LIN {X 0,Y 250.024,Z 759.381,A -85,B 0,C 180,E1 17271.33,E2 17271.33} C_VEL
LIN {X 0,Y 248.705,Z 752.621,A -85,B 0,C 180,E1 17277.4,E2 17277.4} C_VEL
LIN {X 0,Y 248.828,Z 740.046,A -85,B 0,C 180,E1 17283.485,E2 17283.485} C_VEL
LIN {X 0,Y 250.046,Z 721.857,A -85,B 0,C 180,E1 17289.123,E2 17289.123} C_VEL
LIN {X 0,Y 252.287,Z 698.147,A -85,B 0,C 180,E1 17294.071,E2 17294.071} C_VEL
LIN {X 0,Y 254.747,Z 670.659,A -85,B 0,C 180,E1 17297.96,E2 17297.96} C_VEL
LIN {X 0,Y 256.815,Z 639.717,A -85,B 0,C 180,E1 17300.765,E2 17300.765} C_VEL
LIN {X 0,Y 257.718,Z 620.09,A -85,B 0,C 180,E1 17301.928,E2 17301.928} C_VEL
LIN {X 0,Y 260.308,Z 616.482,A -85,B 0,C 180,E1 17302.928,E2 17302.928} C_VEL
LIN {X 0,Y 264.834,Z 607.073,A -85,B 0,C 180,E1 17303.896,E2 17303.896} C_VEL
LIN {X 0,Y 272.961,Z 594.621,A -85,B 0,C 180,E1 17306.378,E2 17306.378} C_VEL
LIN {X 0,Y 281.526,Z 610.071,A -85,B 0,C 180,E1 17312.421,E2 17312.421} C_VEL
LIN {X 0,Y 291.528,Z 631.973,A -85,B 0,C 180,E1 17318.409,E2 17318.409} C_VEL
LIN {X 0,Y 298.079,Z 654.366,A -85,B 0,C 180,E1 17323.266,E2 17323.266} C_VEL
LIN {X 0,Y 299.11,Z 663.186,A -85,B 0,C 180,E1 17324.88,E2 17324.88} C_VEL
LIN {X 0,Y 288.395,Z 696.037,A -85,B 0,C 180,E1 17328.65,E2 17328.65} C_VEL
LIN {X 0,Y 277.431,Z 723.704,A -85,B 0,C 180,E1 17333.247,E2 17333.247} C_VEL
LIN {X 0,Y 266.011,Z 748.871,A -85,B 0,C 180,E1 17339.297,E2 17339.297} C_VEL
LIN {X 0,Y 256.342,Z 769.366,A -85,B 0,C 180,E1 17346.585,E2 17346.585} C_VEL
LIN {X 0,Y 249.921,Z 783.871,A -85,B 0,C 180,E1 17354.413,E2 17354.413} C_VEL
LIN {X 0,Y 246.587,Z 793.255,A -85,B 0,C 180,E1 17362.97,E2 17362.97} C_VEL
LIN {X 0,Y 245.826,Z 796.854,A -85,B 0,C 180,E1 17370.001,E2 17370.001} C_VEL
LIN {X 0,Y 245.618,Z 797.004,A -85,B 0,C 180,E1 17377.059,E2 17377.059} C_VEL
LIN {X 0,Y 246.956,Z 793.586,A -85,B 0,C 180,E1 17384.15,E2 17384.15} C_VEL
LIN {X 0,Y 251.318,Z 784.05,A -85,B 0,C 180,E1 17392.976,E2 17392.976} C_VEL
LIN {X 0,Y 258.612,Z 769.768,A -85,B 0,C 180,E1 17400.706,E2 17400.706} C_VEL
LIN {X 0,Y 269.525,Z 749.005,A -85,B 0,C 180,E1 17408.021,E2 17408.021} C_VEL
LIN {X 0,Y 282.105,Z 723.317,A -85,B 0,C 180,E1 17414.065,E2 17414.065} C_VEL
LIN {X 0,Y 294.764,Z 693.635,A -85,B 0,C 180,E1 17418.777,E2 17418.777} C_VEL
LIN {X 0,Y 304.453,Z 665.385,A -85,B 0,C 180,E1 17421.913,E2 17421.913} C_VEL
LIN {X 0,Y 299.008,Z 642.776,A -85,B 0,C 180,E1 17427.136,E2 17427.136} C_VEL
LIN {X 0,Y 298.518,Z 641.319,A -85,B 0,C 180,E1 17427.506,E2 17427.506} C_VEL
LIN {X 0,Y 282.147,Z 661.718,A -85,B 0,C 180,E1 17429.533,E2 17429.533} C_VEL
LIN {X 0,Y 270.306,Z 673.201,A -85,B 0,C 180,E1 17431.601,E2 17431.601} C_VEL
LIN {X 0,Y 261.762,Z 680.494,A -85,B 0,C 180,E1 17433.454,E2 17433.454} C_VEL
LIN {X 0,Y 258.089,Z 683.189,A -85,B 0,C 180,E1 17434.447,E2 17434.447} C_VEL
LIN {X 0,Y 253.572,Z 685.97,A -85,B 0,C 180,E1 17435.932,E2 17435.932} C_VEL
LIN {X 0,Y 252.951,Z 690.362,A -85,B 0,C 180,E1 17436.705,E2 17436.705} C_VEL
LIN {X 0,Y 250.934,Z 714.808,A -85,B 0,C 180,E1 17440.677,E2 17440.677} C_VEL
LIN {X 0,Y 249.341,Z 734.383,A -85,B 0,C 180,E1 17445.567,E2 17445.567} C_VEL
LIN {X 0,Y 248.688,Z 747.033,A -85,B 0,C 180,E1 17450.386,E2 17450.386} C_VEL
LIN {X 0,Y 248.844,Z 754.316,A -85,B 0,C 180,E1 17454.773,E2 17454.773} C_VEL
LIN {X 0,Y 250.011,Z 758.572,A -85,B 0,C 180,E1 17459.992,E2 17459.992} C_VEL
LIN {X 0,Y 251.473,Z 758.815,A -85,B 0,C 180,E1 17463.432,E2 17463.432} C_VEL
LIN {X 0,Y 255.403,Z 754.257,A -85,B 0,C 180,E1 17469.343,E2 17469.343} C_VEL
LIN {X 0,Y 260.605,Z 743.743,A -85,B 0,C 180,E1 17474.667,E2 17474.667} C_VEL
LIN {X 0,Y 266.042,Z 728.772,A -85,B 0,C 180,E1 17479.027,E2 17479.027} C_VEL
LIN {X 0,Y 271.609,Z 707.895,A -85,B 0,C 180,E1 17482.879,E2 17482.879} C_VEL
LIN {X 0,Y 276.132,Z 682.599,A -85,B 0,C 180,E1 17485.787,E2 17485.787} C_VEL
LIN {X 0,Y 276.83,Z 677.028,A -85,B 0,C 180,E1 17486.267,E2 17486.267} C_VEL
LIN {X 0,Y 282.767,Z 670.413,A -85,B 0,C 180,E1 17487.132,E2 17487.132} C_VEL
LIN {X 0,Y 299.288,Z 647.276,A -85,B 0,C 180,E1 17488.81,E2 17488.81} C_VEL
LIN {X 0,Y 301.073,Z 645.58,A -85,B 0,C 180,E1 17489.104,E2 17489.104} C_VEL
LIN {X 0,Y 309.235,Z 670.823,A -85,B 0,C 180,E1 17494.629,E2 17494.629} C_VEL
LIN {X 0,Y 308.878,Z 675.554,A -85,B 0,C 180,E1 17495.18,E2 17495.18} C_VEL
LIN {X 0,Y 296.991,Z 714.596,A -85,B 0,C 180,E1 17498.62,E2 17498.62} C_VEL
LIN {X 0,Y 284.585,Z 746.683,A -85,B 0,C 180,E1 17502.891,E2 17502.891} C_VEL
LIN {X 0,Y 272.037,Z 774.342,A -85,B 0,C 180,E1 17508.261,E2 17508.261} C_VEL
LIN {X 0,Y 260.443,Z 798.326,A -85,B 0,C 180,E1 17515.094,E2 17515.094} C_VEL
LIN {X 0,Y 251.52,Z 817.448,A -85,B 0,C 180,E1 17523.159,E2 17523.159} C_VEL
LIN {X 0,Y 246.513,Z 831.268,A -85,B 0,C 180,E1 17532.175,E2 17532.175} C_VEL
LIN {X 0,Y 245.059,Z 838.394,A -85,B 0,C 180,E1 17540.101,E2 17540.101} C_VEL
LIN {X 0,Y 244.928,Z 841.087,A -85,B 0,C 180,E1 17546.467,E2 17546.467} C_VEL
LIN {X 0,Y 245.399,Z 841.461,A -85,B 0,C 180,E1 17549.999,E2 17549.999} C_VEL
LIN {X 0,Y 244.964,Z 839.528,A -85,B 0,C 180,E1 17557.077,E2 17557.077} C_VEL
LIN {X 0,Y 246.082,Z 832.265,A -85,B 0,C 180,E1 17566.02,E2 17566.02} C_VEL
LIN {X 0,Y 250.068,Z 819.039,A -85,B 0,C 180,E1 17574.989,E2 17574.989} C_VEL
LIN {X 0,Y 258.016,Z 799.995,A -85,B 0,C 180,E1 17583.254,E2 17583.254} C_VEL
LIN {X 0,Y 268.824,Z 775.778,A -85,B 0,C 180,E1 17590.32,E2 17590.32} C_VEL
LIN {X 0,Y 280.754,Z 747.171,A -85,B 0,C 180,E1 17596.004,E2 17596.004} C_VEL
LIN {X 0,Y 292.476,Z 715.007,A -85,B 0,C 180,E1 17600.354,E2 17600.354} C_VEL
LIN {X 0,Y 297.708,Z 697.847,A -85,B 0,C 180,E1 17602.086,E2 17602.086} C_VEL
LIN {X 0,Y 281.447,Z 707.401,A -85,B 0,C 180,E1 17604.084,E2 17604.084} C_VEL
LIN {X 0,Y 276.293,Z 721.227,A -85,B 0,C 180,E1 17606.569,E2 17606.569} C_VEL
LIN {X 0,Y 268.734,Z 733.756,A -85,B 0,C 180,E1 17608.644,E2 17608.644} C_VEL
LIN {X 0,Y 261.291,Z 743.898,A -85,B 0,C 180,E1 17610.882,E2 17610.882} C_VEL
LIN {X 0,Y 260.962,Z 744.422,A -85,B 0,C 180,E1 17611.073,E2 17611.073} C_VEL
LIN {X 0,Y 253.58,Z 755.494,A -85,B 0,C 180,E1 17616.325,E2 17616.325} C_VEL
LIN {X 0,Y 247.612,Z 761.565,A -85,B 0,C 180,E1 17622.267,E2 17622.267} C_VEL
LIN {X 0,Y 245.037,Z 762.531,A -85,B 0,C 180,E1 17625.748,E2 17625.748} C_VEL
LIN {X 0,Y 242.317,Z 760.769,A -85,B 0,C 180,E1 17631.052,E2 17631.052} C_VEL
LIN {X 0,Y 240.885,Z 753.621,A -85,B 0,C 180,E1 17637.315,E2 17637.315} C_VEL
LIN {X 0,Y 240.963,Z 740.642,A -85,B 0,C 180,E1 17643.599,E2 17643.599} C_VEL
LIN {X 0,Y 242.241,Z 721.934,A -85,B 0,C 180,E1 17649.42,E2 17649.42} C_VEL
LIN {X 0,Y 244.575,Z 697.686,A -85,B 0,C 180,E1 17654.525,E2 17654.525} C_VEL
LIN {X 0,Y 247.222,Z 668.633,A -85,B 0,C 180,E1 17658.594,E2 17658.594} C_VEL
LIN {X 0,Y 249.103,Z 641.736,A -85,B 0,C 180,E1 17661.109,E2 17661.109} C_VEL
LIN {X 0,Y 251.183,Z 639.486,A -85,B 0,C 180,E1 17662.063,E2 17662.063} C_VEL
LIN {X 0,Y 256.836,Z 628.431,A -85,B 0,C 180,E1 17663.259,E2 17663.259} C_VEL
LIN {X 0,Y 258.62,Z 624.905,A -85,B 0,C 180,E1 17663.659,E2 17663.659} C_VEL
LIN {X 0,Y 264.07,Z 614.767,A -85,B 0,C 180,E1 17664.935,E2 17664.935} C_VEL
LIN {X 0,Y 271.122,Z 603.638,A -85,B 0,C 180,E1 17666.882,E2 17666.882} C_VEL
LIN {X 0,Y 279.782,Z 620.232,A -85,B 0,C 180,E1 17673.047,E2 17673.047} C_VEL
LIN {X 0,Y 288.455,Z 642.214,A -85,B 0,C 180,E1 17678.895,E2 17678.895} C_VEL
LIN {X 0,Y 293.409,Z 663.904,A -85,B 0,C 180,E1 17683.625,E2 17683.625} C_VEL
LIN {X 0,Y 283.073,Z 696.013,A -85,B 0,C 180,E1 17687.436,E2 17687.436} C_VEL
LIN {X 0,Y 271.188,Z 724.764,A -85,B 0,C 180,E1 17692.255,E2 17692.255} C_VEL
LIN {X 0,Y 259.284,Z 749.835,A -85,B 0,C 180,E1 17698.41,E2 17698.41} C_VEL
LIN {X 0,Y 249.135,Z 770.237,A -85,B 0,C 180,E1 17705.865,E2 17705.865} C_VEL
LIN {X 0,Y 242.475,Z 784.438,A -85,B 0,C 180,E1 17713.736,E2 17713.736} C_VEL
LIN {X 0,Y 238.773,Z 794.017,A -85,B 0,C 180,E1 17722.738,E2 17722.738} C_VEL
LIN {X 0,Y 237.977,Z 797.575,A -85,B 0,C 180,E1 17730.001,E2 17730.001} C_VEL
LIN {X 0,Y 237.764,Z 797.7,A -85,B 0,C 180,E1 17737.294,E2 17737.294} C_VEL
LIN {X 0,Y 239.24,Z 794.261,A -85,B 0,C 180,E1 17744.616,E2 17744.616} C_VEL
LIN {X 0,Y 243.928,Z 784.719,A -85,B 0,C 180,E1 17753.714,E2 17753.714} C_VEL
LIN {X 0,Y 251.718,Z 770.414,A -85,B 0,C 180,E1 17761.643,E2 17761.643} C_VEL
LIN {X 0,Y 263.246,Z 749.644,A -85,B 0,C 180,E1 17769.097,E2 17769.097} C_VEL
LIN {X 0,Y 276.418,Z 723.92,A -85,B 0,C 180,E1 17775.217,E2 17775.217} C_VEL
LIN {X 0,Y 289.272,Z 695.04,A -85,B 0,C 180,E1 17779.849,E2 17779.849} C_VEL
LIN {X 0,Y 298.783,Z 668.445,A -85,B 0,C 180,E1 17782.891,E2 17782.891} C_VEL
LIN {X 0,Y 295.453,Z 652.057,A -85,B 0,C 180,E1 17786.775,E2 17786.775} C_VEL
LIN {X 0,Y 280.732,Z 668.46,A -85,B 0,C 180,E1 17788.597,E2 17788.597} C_VEL
LIN {X 0,Y 268.852,Z 679.276,A -85,B 0,C 180,E1 17790.577,E2 17790.577} C_VEL
LIN {X 0,Y 260.135,Z 686.335,A -85,B 0,C 180,E1 17792.341,E2 17792.341} C_VEL
LIN {X 0,Y 247.479,Z 695.108,A -85,B 0,C 180,E1 17795.816,E2 17795.816} C_VEL
LIN {X 0,Y 244.805,Z 696.846,A -85,B 0,C 180,E1 17797.215,E2 17797.215} C_VEL
LIN {X 0,Y 242.653,Z 719.9,A -85,B 0,C 180,E1 17801.406,E2 17801.406} C_VEL
LIN {X 0,Y 241.28,Z 738.13,A -85,B 0,C 180,E1 17806.427,E2 17806.427} C_VEL
LIN {X 0,Y 240.793,Z 750.869,A -85,B 0,C 180,E1 17811.886,E2 17811.886} C_VEL
LIN {X 0,Y 241.623,Z 758.616,A -85,B 0,C 180,E1 17817.97,E2 17817.97} C_VEL
LIN {X 0,Y 243.765,Z 760.451,A -85,B 0,C 180,E1 17823.541,E2 17823.541} C_VEL
LIN {X 0,Y 247.928,Z 756.572,A -85,B 0,C 180,E1 17829.627,E2 17829.627} C_VEL
LIN {X 0,Y 253.445,Z 746.827,A -85,B 0,C 180,E1 17835.091,E2 17835.091} C_VEL
LIN {X 0,Y 259.82,Z 731.185,A -85,B 0,C 180,E1 17839.943,E2 17839.943} C_VEL
LIN {X 0,Y 265.992,Z 710.335,A -85,B 0,C 180,E1 17843.945,E2 17843.945} C_VEL
LIN {X 0,Y 270.352,Z 689.796,A -85,B 0,C 180,E1 17846.514,E2 17846.514} C_VEL
LIN {X 0,Y 276.719,Z 683.522,A -85,B 0,C 180,E1 17847.48,E2 17847.48} C_VEL
LIN {X 0,Y 292.53,Z 664.243,A -85,B 0,C 180,E1 17849.263,E2 17849.263} C_VEL
LIN {X 0,Y 297.533,Z 656.963,A -85,B 0,C 180,E1 17849.663,E2 17849.663} C_VEL
LIN {X 0,Y 300.096,Z 661.994,A -85,B 0,C 180,E1 17851.101,E2 17851.101} C_VEL
LIN {X 0,Y 303.842,Z 675.889,A -85,B 0,C 180,E1 17854.044,E2 17854.044} C_VEL
LIN {X 0,Y 291.982,Z 713.613,A -85,B 0,C 180,E1 17857.373,E2 17857.373} C_VEL
LIN {X 0,Y 279.227,Z 745.459,A -85,B 0,C 180,E1 17861.604,E2 17861.604} C_VEL
LIN {X 0,Y 265.928,Z 773.501,A -85,B 0,C 180,E1 17867.076,E2 17867.076} C_VEL
LIN {X 0,Y 253.719,Z 797.558,A -85,B 0,C 180,E1 17874.027,E2 17874.027} C_VEL
LIN {X 0,Y 244.173,Z 816.877,A -85,B 0,C 180,E1 17882.382,E2 17882.382} C_VEL
LIN {X 0,Y 238.791,Z 830.549,A -85,B 0,C 180,E1 17891.578,E2 17891.578} C_VEL
LIN {X 0,Y 237.146,Z 837.999,A -85,B 0,C 180,E1 17900.254,E2 17900.254} C_VEL
LIN {X 0,Y 237.044,Z 840.385,A -85,B 0,C 180,E1 17906.349,E2 17906.349} C_VEL
LIN {X 0,Y 237.516,Z 840.75,A -85,B 0,C 180,E1 17909.999,E2 17909.999} C_VEL
LIN {X 0,Y 237.073,Z 838.786,A -85,B 0,C 180,E1 17917.314,E2 17917.314} C_VEL
LIN {X 0,Y 237.855,Z 833.399,A -85,B 0,C 180,E1 17924.702,E2 17924.702} C_VEL
LIN {X 0,Y 241.457,Z 821.32,A -85,B 0,C 180,E1 17933.97,E2 17933.97} C_VEL
LIN {X 0,Y 248.933,Z 803.637,A -85,B 0,C 180,E1 17942.536,E2 17942.536} C_VEL
LIN {X 0,Y 259.384,Z 781.296,A -85,B 0,C 180,E1 17949.792,E2 17949.792} C_VEL
LIN {X 0,Y 271.8,Z 753.577,A -85,B 0,C 180,E1 17955.918,E2 17955.918} C_VEL
LIN {X 0,Y 284.241,Z 722.074,A -85,B 0,C 180,E1 17960.616,E2 17960.616} C_VEL
LIN {X 0,Y 287.935,Z 711.502,A -85,B 0,C 180,E1 17961.832,E2 17961.832} C_VEL
LIN {X 0,Y 287.56,Z 710.09,A -85,B 0,C 180,E1 17962.155,E2 17962.155} C_VEL
LIN {X 0,Y 274.608,Z 716.397,A -85,B 0,C 180,E1 17963.919,E2 17963.919} C_VEL
LIN {X 0,Y 264.992,Z 737.124,A -85,B 0,C 180,E1 17968.679,E2 17968.679} C_VEL
LIN {X 0,Y 260.962,Z 744.422,A -85,B 0,C 180,E1 17971.073,E2 17971.073} C_VEL
LIN {X 0,Y 252.831,Z 753.354,A -85,B 0,C 180,E1 17973.932,E2 17973.932} C_VEL
LIN {X 0,Y 245.199,Z 759.728,A -85,B 0,C 180,E1 17976.926,E2 17976.926} C_VEL
LIN {X 0,Y 244.902,Z 759.939,A -85,B 0,C 180,E1 17977.162,E2 17977.162} C_VEL
LIN {X 0,Y 240.338,Z 763.539,A -85,B 0,C 180,E1 17981.712,E2 17981.712} C_VEL
LIN {X 0,Y 237.568,Z 764.279,A -85,B 0,C 180,E1 17985.29,E2 17985.29} C_VEL
LIN {X 0,Y 234.625,Z 762.124,A -85,B 0,C 180,E1 17990.756,E2 17990.756} C_VEL
LIN {X 0,Y 233.035,Z 754.61,A -85,B 0,C 180,E1 17997.225,E2 17997.225} C_VEL
LIN {X 0,Y 233.093,Z 741.101,A -85,B 0,C 180,E1 18003.72,E2 18003.72} C_VEL
LIN {X 0,Y 234.445,Z 721.899,A -85,B 0,C 180,E1 18009.736,E2 18009.736} C_VEL
LIN {X 0,Y 236.758,Z 698.18,A -85,B 0,C 180,E1 18014.779,E2 18014.779} C_VEL
LIN {X 0,Y 239.462,Z 669.534,A -85,B 0,C 180,E1 18018.897,E2 18018.897} C_VEL
LIN {X 0,Y 240.33,Z 659.681,A -85,B 0,C 180,E1 18020.072,E2 18020.072} C_VEL
LIN {X 0,Y 243.745,Z 655.911,A -85,B 0,C 180,E1 18021.494,E2 18021.494} C_VEL
LIN {X 0,Y 248.777,Z 647.551,A -85,B 0,C 180,E1 18022.619,E2 18022.619} C_VEL
LIN {X 0,Y 254.503,Z 639.221,A -85,B 0,C 180,E1 18024.229,E2 18024.229} C_VEL
LIN {X 0,Y 260.251,Z 628.282,A -85,B 0,C 180,E1 18025.326,E2 18025.326} C_VEL
LIN {X 0,Y 267.14,Z 616.064,A -85,B 0,C 180,E1 18026.874,E2 18026.874} C_VEL
LIN {X 0,Y 269.344,Z 613.016,A -85,B 0,C 180,E1 18027.512,E2 18027.512} C_VEL
LIN {X 0,Y 277.59,Z 630.287,A -85,B 0,C 180,E1 18033.585,E2 18033.585} C_VEL
LIN {X 0,Y 284.434,Z 650.554,A -85,B 0,C 180,E1 18038.986,E2 18038.986} C_VEL
LIN {X 0,Y 287.585,Z 668.623,A -85,B 0,C 180,E1 18042.956,E2 18042.956} C_VEL
LIN {X 0,Y 275.911,Z 700.839,A -85,B 0,C 180,E1 18046.865,E2 18046.865} C_VEL
LIN {X 0,Y 263.358,Z 729.318,A -85,B 0,C 180,E1 18051.974,E2 18051.974} C_VEL
LIN {X 0,Y 251.216,Z 753.431,A -85,B 0,C 180,E1 18058.288,E2 18058.288} C_VEL
LIN {X 0,Y 240.94,Z 773.175,A -85,B 0,C 180,E1 18066.059,E2 18066.059} C_VEL
LIN {X 0,Y 233.81,Z 787.611,A -85,B 0,C 180,E1 18075.038,E2 18075.038} C_VEL
LIN {X 0,Y 230.969,Z 794.774,A -85,B 0,C 180,E1 18082.492,E2 18082.492} C_VEL
LIN {X 0,Y 230.122,Z 798.296,A -85,B 0,C 180,E1 18090.001,E2 18090.001} C_VEL
LIN {X 0,Y 229.925,Z 798.396,A -85,B 0,C 180,E1 18097.544,E2 18097.544} C_VEL
LIN {X 0,Y 231.529,Z 794.941,A -85,B 0,C 180,E1 18105.114,E2 18105.114} C_VEL
LIN {X 0,Y 236.582,Z 785.381,A -85,B 0,C 180,E1 18114.498,E2 18114.498} C_VEL
LIN {X 0,Y 244.907,Z 771.067,A -85,B 0,C 180,E1 18122.63,E2 18122.63} C_VEL
LIN {X 0,Y 257.095,Z 750.279,A -85,B 0,C 180,E1 18130.22,E2 18130.22} C_VEL
LIN {X 0,Y 270.864,Z 724.529,A -85,B 0,C 180,E1 18136.413,E2 18136.413} C_VEL
LIN {X 0,Y 284.529,Z 694.748,A -85,B 0,C 180,E1 18141.199,E2 18141.199} C_VEL
LIN {X 0,Y 293.095,Z 671.056,A -85,B 0,C 180,E1 18144.012,E2 18144.012} C_VEL
LIN {X 0,Y 291.882,Z 663.652,A -85,B 0,C 180,E1 18145.821,E2 18145.821} C_VEL
LIN {X 0,Y 290.566,Z 663.826,A -85,B 0,C 180,E1 18146.205,E2 18146.205} C_VEL
LIN {X 0,Y 273.557,Z 680.347,A -85,B 0,C 180,E1 18148.387,E2 18148.387} C_VEL
LIN {X 0,Y 258.118,Z 692.28,A -85,B 0,C 180,E1 18151.287,E2 18151.287} C_VEL
LIN {X 0,Y 244.499,Z 701.239,A -85,B 0,C 180,E1 18154.894,E2 18154.894} C_VEL
LIN {X 0,Y 236.5,Z 705.475,A -85,B 0,C 180,E1 18157.975,E2 18157.975} C_VEL
LIN {X 0,Y 233.928,Z 731.79,A -85,B 0,C 180,E1 18164.079,E2 18164.079} C_VEL
LIN {X 0,Y 233.019,Z 747.465,A -85,B 0,C 180,E1 18169.733,E2 18169.733} C_VEL
LIN {X 0,Y 233.262,Z 756.973,A -85,B 0,C 180,E1 18175.353,E2 18175.353} C_VEL
LIN {X 0,Y 234.413,Z 761.088,A -85,B 0,C 180,E1 18179.992,E2 18179.992} C_VEL
LIN {X 0,Y 236.034,Z 762.072,A -85,B 0,C 180,E1 18183.657,E2 18183.657} C_VEL
LIN {X 0,Y 239.713,Z 759.701,A -85,B 0,C 180,E1 18189.046,E2 18189.046} C_VEL
LIN {X 0,Y 244.85,Z 752.504,A -85,B 0,C 180,E1 18194.264,E2 18194.264} C_VEL
LIN {X 0,Y 251.283,Z 739.619,A -85,B 0,C 180,E1 18199.278,E2 18199.278} C_VEL
LIN {X 0,Y 258.195,Z 720.933,A -85,B 0,C 180,E1 18203.683,E2 18203.683} C_VEL
LIN {X 0,Y 264.036,Z 700.867,A -85,B 0,C 180,E1 18206.797,E2 18206.797} C_VEL
LIN {X 0,Y 278.176,Z 687.826,A -85,B 0,C 180,E1 18208.816,E2 18208.816} C_VEL
LIN {X 0,Y 295.409,Z 668.152,A -85,B 0,C 180,E1 18210.711,E2 18210.711} C_VEL
LIN {X 0,Y 298.099,Z 678.398,A -85,B 0,C 180,E1 18212.973,E2 18212.973} C_VEL
LIN {X 0,Y 286.43,Z 714.509,A -85,B 0,C 180,E1 18216.283,E2 18216.283} C_VEL
LIN {X 0,Y 273.163,Z 746.055,A -85,B 0,C 180,E1 18220.564,E2 18220.564} C_VEL
LIN {X 0,Y 259.341,Z 773.788,A -85,B 0,C 180,E1 18226.108,E2 18226.108} C_VEL
LIN {X 0,Y 246.427,Z 797.976,A -85,B 0,C 180,E1 18233.336,E2 18233.336} C_VEL
LIN {X 0,Y 236.934,Z 816.142,A -85,B 0,C 180,E1 18241.463,E2 18241.463} C_VEL
LIN {X 0,Y 231.088,Z 829.825,A -85,B 0,C 180,E1 18250.94,E2 18250.94} C_VEL
LIN {X 0,Y 229.407,Z 836.487,A -85,B 0,C 180,E1 18258.617,E2 18258.617} C_VEL
LIN {X 0,Y 229.149,Z 839.681,A -85,B 0,C 180,E1 18266.223,E2 18266.223} C_VEL
LIN {X 0,Y 229.655,Z 840.042,A -85,B 0,C 180,E1 18269.999,E2 18269.999} C_VEL
LIN {X 0,Y 229.274,Z 837.177,A -85,B 0,C 180,E1 18279.208,E2 18279.208} C_VEL
LIN {X 0,Y 230.872,Z 829.6,A -85,B 0,C 180,E1 18288.089,E2 18288.089} C_VEL
LIN {X 0,Y 236.058,Z 815.529,A -85,B 0,C 180,E1 18297.613,E2 18297.613} C_VEL
LIN {X 0,Y 245.568,Z 795.534,A -85,B 0,C 180,E1 18306.264,E2 18306.264} C_VEL
LIN {X 0,Y 257.437,Z 771.15,A -85,B 0,C 180,E1 18313.276,E2 18313.276} C_VEL
LIN {X 0,Y 270.419,Z 742.338,A -85,B 0,C 180,E1 18318.887,E2 18318.887} C_VEL
LIN {X 0,Y 279.37,Z 719.677,A -85,B 0,C 180,E1 18322.034,E2 18322.034} C_VEL
LIN {X 0,Y 267.779,Z 724.681,A -85,B 0,C 180,E1 18323.731,E2 18323.731} C_VEL
LIN {X 0,Y 257.392,Z 743.475,A -85,B 0,C 180,E1 18328.736,E2 18328.736} C_VEL
LIN {X 0,Y 249.093,Z 755.381,A -85,B 0,C 180,E1 18333.955,E2 18333.955} C_VEL
LIN {X 0,Y 244.902,Z 759.939,A -85,B 0,C 180,E1 18337.162,E2 18337.162} C_VEL
LIN {X 0,Y 237.215,Z 764.301,A -85,B 0,C 180,E1 18340.775,E2 18340.775} C_VEL
LIN {X 0,Y 230.648,Z 766.018,A -85,B 0,C 180,E1 18344.137,E2 18344.137} C_VEL
LIN {X 0,Y 230.188,Z 766.002,A -85,B 0,C 180,E1 18344.667,E2 18344.667} C_VEL
LIN {X 0,Y 226.927,Z 763.456,A -85,B 0,C 180,E1 18350.439,E2 18350.439} C_VEL
LIN {X 0,Y 225.198,Z 755.513,A -85,B 0,C 180,E1 18357.128,E2 18357.128} C_VEL
LIN {X 0,Y 225.249,Z 741.548,A -85,B 0,C 180,E1 18363.85,E2 18363.85} C_VEL
LIN {X 0,Y 226.658,Z 721.715,A -85,B 0,C 180,E1 18370.074,E2 18370.074} C_VEL
LIN {X 0,Y 229.099,Z 697.318,A -85,B 0,C 180,E1 18375.285,E2 18375.285} C_VEL
LIN {X 0,Y 231.429,Z 674.968,A -85,B 0,C 180,E1 18378.79,E2 18378.79} C_VEL
LIN {X 0,Y 234.275,Z 672.171,A -85,B 0,C 180,E1 18380.19,E2 18380.19} C_VEL
LIN {X 0,Y 239.358,Z 665.362,A -85,B 0,C 180,E1 18381.582,E2 18381.582} C_VEL
LIN {X 0,Y 244.683,Z 658.9,A -85,B 0,C 180,E1 18383.28,E2 18383.28} C_VEL
LIN {X 0,Y 249.02,Z 652.308,A -85,B 0,C 180,E1 18384.153,E2 18384.153} C_VEL
LIN {X 0,Y 255.599,Z 642.86,A -85,B 0,C 180,E1 18385.783,E2 18385.783} C_VEL
LIN {X 0,Y 261.78,Z 631.865,A -85,B 0,C 180,E1 18386.881,E2 18386.881} C_VEL
LIN {X 0,Y 266.729,Z 622.841,A -85,B 0,C 180,E1 18387.832,E2 18387.832} C_VEL
LIN {X 0,Y 268.523,Z 624.772,A -85,B 0,C 180,E1 18389.001,E2 18389.001} C_VEL
LIN {X 0,Y 275.979,Z 643.338,A -85,B 0,C 180,E1 18395.046,E2 18395.046} C_VEL
LIN {X 0,Y 281.26,Z 664.991,A -85,B 0,C 180,E1 18400.558,E2 18400.558} C_VEL
LIN {X 0,Y 281.899,Z 671.385,A -85,B 0,C 180,E1 18401.945,E2 18401.945} C_VEL
LIN {X 0,Y 269.792,Z 703.206,A -85,B 0,C 180,E1 18405.915,E2 18405.915} C_VEL
LIN {X 0,Y 257.222,Z 730.375,A -85,B 0,C 180,E1 18410.897,E2 18410.897} C_VEL
LIN {X 0,Y 244.582,Z 754.383,A -85,B 0,C 180,E1 18417.323,E2 18417.323} C_VEL
LIN {X 0,Y 233.562,Z 774.414,A -85,B 0,C 180,E1 18425.463,E2 18425.463} C_VEL
LIN {X 0,Y 226.198,Z 788.417,A -85,B 0,C 180,E1 18434.522,E2 18434.522} C_VEL
LIN {X 0,Y 223.178,Z 795.53,A -85,B 0,C 180,E1 18442.228,E2 18442.228} C_VEL
LIN {X 0,Y 222.245,Z 799.019,A -85,B 0,C 180,E1 18450.001,E2 18450.001} C_VEL
LIN {X 0,Y 222.094,Z 799.091,A -85,B 0,C 180,E1 18457.812,E2 18457.812} C_VEL
LIN {X 0,Y 223.841,Z 795.617,A -85,B 0,C 180,E1 18465.646,E2 18465.646} C_VEL
LIN {X 0,Y 229.279,Z 786.041,A -85,B 0,C 180,E1 18475.332,E2 18475.332} C_VEL
LIN {X 0,Y 238.165,Z 771.732,A -85,B 0,C 180,E1 18483.674,E2 18483.674} C_VEL
LIN {X 0,Y 251.034,Z 750.91,A -85,B 0,C 180,E1 18491.4,E2 18491.4} C_VEL
LIN {X 0,Y 265.446,Z 725.168,A -85,B 0,C 180,E1 18497.656,E2 18497.656} C_VEL
LIN {X 0,Y 279.578,Z 695.439,A -85,B 0,C 180,E1 18502.453,E2 18502.453} C_VEL
LIN {X 0,Y 287.531,Z 674.463,A -85,B 0,C 180,E1 18504.981,E2 18504.981} C_VEL
LIN {X 0,Y 287.421,Z 673.561,A -85,B 0,C 180,E1 18505.215,E2 18505.215} C_VEL
LIN {X 0,Y 261.024,Z 694.856,A -85,B 0,C 180,E1 18509.166,E2 18509.166} C_VEL
LIN {X 0,Y 241.148,Z 707.313,A -85,B 0,C 180,E1 18514.012,E2 18514.012} C_VEL
LIN {X 0,Y 227.965,Z 714.215,A -85,B 0,C 180,E1 18519.156,E2 18519.156} C_VEL
LIN {X 0,Y 227.518,Z 716.023,A -85,B 0,C 180,E1 18519.87,E2 18519.87} C_VEL
LIN {X 0,Y 225.788,Z 736.58,A -85,B 0,C 180,E1 18525.228,E2 18525.228} C_VEL
LIN {X 0,Y 225.111,Z 751.52,A -85,B 0,C 180,E1 18531.316,E2 18531.316} C_VEL
LIN {X 0,Y 225.776,Z 759.991,A -85,B 0,C 180,E1 18537.214,E2 18537.214} C_VEL
LIN {X 0,Y 228.297,Z 763.608,A -85,B 0,C 180,E1 18543.781,E2 18543.781} C_VEL
LIN {X 0,Y 232.182,Z 761.855,A -85,B 0,C 180,E1 18549.342,E2 18549.342} C_VEL
LIN {X 0,Y 237.647,Z 755.361,A -85,B 0,C 180,E1 18554.705,E2 18554.705} C_VEL
LIN {X 0,Y 244.459,Z 743.424,A -85,B 0,C 180,E1 18559.839,E2 18559.839} C_VEL
LIN {X 0,Y 252.185,Z 725.139,A -85,B 0,C 180,E1 18564.519,E2 18564.519} C_VEL
LIN {X 0,Y 257.266,Z 711.17,A -85,B 0,C 180,E1 18567.03,E2 18567.03} C_VEL
LIN {X 0,Y 274.815,Z 697.114,A -85,B 0,C 180,E1 18569.609,E2 18569.609} C_VEL
LIN {X 0,Y 290.994,Z 679.447,A -85,B 0,C 180,E1 18571.229,E2 18571.229} C_VEL
LIN {X 0,Y 292.311,Z 681.194,A -85,B 0,C 180,E1 18571.884,E2 18571.884} C_VEL
LIN {X 0,Y 280.897,Z 715.509,A -85,B 0,C 180,E1 18575.166,E2 18575.166} C_VEL
LIN {X 0,Y 267.368,Z 746.253,A -85,B 0,C 180,E1 18579.411,E2 18579.411} C_VEL
LIN {X 0,Y 252.435,Z 774.877,A -85,B 0,C 180,E1 18585.295,E2 18585.295} C_VEL
LIN {X 0,Y 239.189,Z 798.396,A -85,B 0,C 180,E1 18592.605,E2 18592.605} C_VEL
LIN {X 0,Y 228.894,Z 817.058,A -85,B 0,C 180,E1 18601.443,E2 18601.443} C_VEL
LIN {X 0,Y 223.059,Z 830.112,A -85,B 0,C 180,E1 18611.256,E2 18611.256} C_VEL
LIN {X 0,Y 221.335,Z 837.087,A -85,B 0,C 180,E1 18620.562,E2 18620.562} C_VEL
LIN {X 0,Y 221.77,Z 839.33,A -85,B 0,C 180,E1 18629.999,E2 18629.999} C_VEL
LIN {X 0,Y 221.396,Z 836.425,A -85,B 0,C 180,E1 18639.539,E2 18639.539} C_VEL
LIN {X 0,Y 223.176,Z 828.677,A -85,B 0,C 180,E1 18648.832,E2 18648.832} C_VEL
LIN {X 0,Y 228.782,Z 814.607,A -85,B 0,C 180,E1 18658.571,E2 18658.571} C_VEL
LIN {X 0,Y 238.789,Z 794.744,A -85,B 0,C 180,E1 18667.357,E2 18667.357} C_VEL
LIN {X 0,Y 251.036,Z 770.828,A -85,B 0,C 180,E1 18674.374,E2 18674.374} C_VEL
LIN {X 0,Y 264.558,Z 742.154,A -85,B 0,C 180,E1 18680.044,E2 18680.044} C_VEL
LIN {X 0,Y 269.825,Z 729.147,A -85,B 0,C 180,E1 18682.044,E2 18682.044} C_VEL
LIN {X 0,Y 261.11,Z 731.955,A -85,B 0,C 180,E1 18683.428,E2 18683.428} C_VEL
LIN {X 0,Y 250.763,Z 747.984,A -85,B 0,C 180,E1 18688.236,E2 18688.236} C_VEL
LIN {X 0,Y 241.205,Z 759.465,A -85,B 0,C 180,E1 18694.037,E2 18694.037} C_VEL
LIN {X 0,Y 235.304,Z 764.408,A -85,B 0,C 180,E1 18698.82,E2 18698.82} C_VEL
LIN {X 0,Y 230.188,Z 766.002,A -85,B 0,C 180,E1 18704.667,E2 18704.667} C_VEL
LIN {X 0,Y 225.75,Z 765.698,A -85,B 0,C 180,E1 18707.773,E2 18707.773} C_VEL
LIN {X 0,Y 218.412,Z 762.484,A -85,B 0,C 180,E1 18712.46,E2 18712.46} C_VEL
LIN {X 0,Y 218.153,Z 761.875,A -85,B 0,C 180,E1 18713.013,E2 18713.013} C_VEL
LIN {X 0,Y 217.13,Z 750.927,A -85,B 0,C 180,E1 18720.009,E2 18720.009} C_VEL
LIN {X 0,Y 217.731,Z 734.966,A -85,B 0,C 180,E1 18726.476,E2 18726.476} C_VEL
LIN {X 0,Y 219.797,Z 712.246,A -85,B 0,C 180,E1 18732.65,E2 18732.65} C_VEL
LIN {X 0,Y 222.351,Z 688.426,A -85,B 0,C 180,E1 18737.263,E2 18737.263} C_VEL
LIN {X 0,Y 225.708,Z 685.309,A -85,B 0,C 180,E1 18739.012,E2 18739.012} C_VEL
LIN {X 0,Y 236.485,Z 673.075,A -85,B 0,C 180,E1 18742.52,E2 18742.52} C_VEL
LIN {X 0,Y 246.051,Z 661.511,A -85,B 0,C 180,E1 18745.067,E2 18745.067} C_VEL
LIN {X 0,Y 257.731,Z 644.998,A -85,B 0,C 180,E1 18747.466,E2 18747.466} C_VEL
LIN {X 0,Y 264.574,Z 633.572,A -85,B 0,C 180,E1 18748.633,E2 18748.633} C_VEL
LIN {X 0,Y 265.409,Z 632.409,A -85,B 0,C 180,E1 18748.831,E2 18748.831} C_VEL
LIN {X 0,Y 272.038,Z 650.833,A -85,B 0,C 180,E1 18754.926,E2 18754.926} C_VEL
LIN {X 0,Y 276.078,Z 671.501,A -85,B 0,C 180,E1 18760.297,E2 18760.297} C_VEL
LIN {X 0,Y 275.342,Z 676.73,A -85,B 0,C 180,E1 18761.183,E2 18761.183} C_VEL
LIN {X 0,Y 262.178,Z 708.882,A -85,B 0,C 180,E1 18765.449,E2 18765.449} C_VEL
LIN {X 0,Y 248.542,Z 736.503,A -85,B 0,C 180,E1 18770.952,E2 18770.952} C_VEL
LIN {X 0,Y 235.153,Z 760.276,A -85,B 0,C 180,E1 18778.031,E2 18778.031} C_VEL
LIN {X 0,Y 224.689,Z 778.162,A -85,B 0,C 180,E1 18786.235,E2 18786.235} C_VEL
LIN {X 0,Y 217.735,Z 790.951,A -85,B 0,C 180,E1 18795.583,E2 18795.583} C_VEL
LIN {X 0,Y 214.99,Z 797.471,A -85,B 0,C 180,E1 18803.957,E2 18803.957} C_VEL
LIN {X 0,Y 214.389,Z 799.741,A -85,B 0,C 180,E1 18810.001,E2 18810.001} C_VEL
LIN {X 0,Y 214.261,Z 799.787,A -85,B 0,C 180,E1 18818.099,E2 18818.099} C_VEL
LIN {X 0,Y 216.164,Z 796.3,A -85,B 0,C 180,E1 18826.217,E2 18826.217} C_VEL
LIN {X 0,Y 222.029,Z 786.703,A -85,B 0,C 180,E1 18836.221,E2 18836.221} C_VEL
LIN {X 0,Y 231.533,Z 772.381,A -85,B 0,C 180,E1 18844.775,E2 18844.775} C_VEL
LIN {X 0,Y 245.081,Z 751.571,A -85,B 0,C 180,E1 18852.639,E2 18852.639} C_VEL
LIN {X 0,Y 260.139,Z 725.786,A -85,B 0,C 180,E1 18858.955,E2 18858.955} C_VEL
LIN {X 0,Y 274.897,Z 695.835,A -85,B 0,C 180,E1 18863.797,E2 18863.797} C_VEL
LIN {X 0,Y 279.5,Z 684.983,A -85,B 0,C 180,E1 18865.127,E2 18865.127} C_VEL
LIN {X 0,Y 267.224,Z 694.814,A -85,B 0,C 180,E1 18866.734,E2 18866.734} C_VEL
LIN {X 0,Y 249.28,Z 706.815,A -85,B 0,C 180,E1 18870.029,E2 18870.029} C_VEL
LIN {X 0,Y 227.694,Z 718.455,A -85,B 0,C 180,E1 18876.559,E2 18876.559} C_VEL
LIN {X 0,Y 220.174,Z 722.202,A -85,B 0,C 180,E1 18879.95,E2 18879.95} C_VEL
LIN {X 0,Y 219.002,Z 723.17,A -85,B 0,C 180,E1 18881.147,E2 18881.147} C_VEL
LIN {X 0,Y 217.676,Z 740.922,A -85,B 0,C 180,E1 18886.395,E2 18886.395} C_VEL
LIN {X 0,Y 217.305,Z 755.257,A -85,B 0,C 180,E1 18893.011,E2 18893.011} C_VEL
LIN {X 0,Y 218.758,Z 763.34,A -85,B 0,C 180,E1 18899.991,E2 18899.991} C_VEL
LIN {X 0,Y 220.545,Z 765.109,A -85,B 0,C 180,E1 18903.914,E2 18903.914} C_VEL
LIN {X 0,Y 224.649,Z 763.963,A -85,B 0,C 180,E1 18909.659,E2 18909.659} C_VEL
LIN {X 0,Y 230.46,Z 758.165,A -85,B 0,C 180,E1 18915.175,E2 18915.175} C_VEL
LIN {X 0,Y 238.334,Z 745.978,A -85,B 0,C 180,E1 18920.855,E2 18920.855} C_VEL
LIN {X 0,Y 246.248,Z 729.346,A -85,B 0,C 180,E1 18925.393,E2 18925.393} C_VEL
LIN {X 0,Y 250.672,Z 720.32,A -85,B 0,C 180,E1 18927.315,E2 18927.315} C_VEL
LIN {X 0,Y 269.872,Z 706.887,A -85,B 0,C 180,E1 18930.207,E2 18930.207} C_VEL
LIN {X 0,Y 284.007,Z 694.138,A -85,B 0,C 180,E1 18931.763,E2 18931.763} C_VEL
LIN {X 0,Y 270.584,Z 727.642,A -85,B 0,C 180,E1 18935.353,E2 18935.353} C_VEL
LIN {X 0,Y 255.817,Z 757.713,A -85,B 0,C 180,E1 18940.272,E2 18940.272} C_VEL
LIN {X 0,Y 241.222,Z 783.321,A -85,B 0,C 180,E1 18946.511,E2 18946.511} C_VEL
LIN {X 0,Y 228.436,Z 804.595,A -85,B 0,C 180,E1 18954.3,E2 18954.3} C_VEL
LIN {X 0,Y 219.294,Z 820.903,A -85,B 0,C 180,E1 18963.433,E2 18963.433} C_VEL
LIN {X 0,Y 214.436,Z 832.177,A -85,B 0,C 180,E1 18973.649,E2 18973.649} C_VEL
LIN {X 0,Y 213.398,Z 837.127,A -85,B 0,C 180,E1 18981.868,E2 18981.868} C_VEL
LIN {X 0,Y 213.907,Z 838.621,A -85,B 0,C 180,E1 18989.999,E2 18989.999} C_VEL
LIN {X 0,Y 213.551,Z 835.629,A -85,B 0,C 180,E1 18999.97,E2 18999.97} C_VEL
LIN {X 0,Y 215.39,Z 828.165,A -85,B 0,C 180,E1 19009.246,E2 19009.246} C_VEL
LIN {X 0,Y 221.605,Z 813.692,A -85,B 0,C 180,E1 19019.586,E2 19019.586} C_VEL
LIN {X 0,Y 231.85,Z 794.451,A -85,B 0,C 180,E1 19028.318,E2 19028.318} C_VEL
LIN {X 0,Y 244.788,Z 770.419,A -85,B 0,C 180,E1 19035.551,E2 19035.551} C_VEL
LIN {X 0,Y 259.033,Z 741.432,A -85,B 0,C 180,E1 19041.344,E2 19041.344} C_VEL
LIN {X 0,Y 260.587,Z 737.236,A -85,B 0,C 180,E1 19042.09,E2 19042.09} C_VEL
LIN {X 0,Y 254.208,Z 739.018,A -85,B 0,C 180,E1 19043.135,E2 19043.135} C_VEL
LIN {X 0,Y 243.18,Z 753.444,A -85,B 0,C 180,E1 19048.176,E2 19048.176} C_VEL
LIN {X 0,Y 234.574,Z 762.203,A -85,B 0,C 180,E1 19053.246,E2 19053.246} C_VEL
LIN {X 0,Y 229.662,Z 765.81,A -85,B 0,C 180,E1 19056.922,E2 19056.922} C_VEL
LIN {X 0,Y 225.86,Z 767.565,A -85,B 0,C 180,E1 19060.494,E2 19060.494} C_VEL
LIN {X 0,Y 222.593,Z 767.672,A -85,B 0,C 180,E1 19064.33,E2 19064.33} C_VEL
LIN {X 0,Y 219.211,Z 764.772,A -85,B 0,C 180,E1 19070.099,E2 19070.099} C_VEL
LIN {X 0,Y 218.153,Z 761.875,A -85,B 0,C 180,E1 19073.013,E2 19073.013} C_VEL
LIN {X 0,Y 214.981,Z 757.821,A -85,B 0,C 180,E1 19076.209,E2 19076.209} C_VEL
LIN {X 0,Y 209.35,Z 749.709,A -85,B 0,C 180,E1 19080.866,E2 19080.866} C_VEL
LIN {X 0,Y 209.239,Z 748.581,A -85,B 0,C 180,E1 19081.389,E2 19081.389} C_VEL
LIN {X 0,Y 210.3,Z 730.058,A -85,B 0,C 180,E1 19088.261,E2 19088.261} C_VEL
LIN {X 0,Y 212.537,Z 706.831,A -85,B 0,C 180,E1 19094.136,E2 19094.136} C_VEL
LIN {X 0,Y 213.26,Z 700.61,A -85,B 0,C 180,E1 19095.397,E2 19095.397} C_VEL
LIN {X 0,Y 217.158,Z 697.044,A -85,B 0,C 180,E1 19097.689,E2 19097.689} C_VEL
LIN {X 0,Y 225.457,Z 688.695,A -85,B 0,C 180,E1 19100.946,E2 19100.946} C_VEL
LIN {X 0,Y 235.612,Z 678.013,A -85,B 0,C 180,E1 19104.008,E2 19104.008} C_VEL
LIN {X 0,Y 245.8,Z 666.487,A -85,B 0,C 180,E1 19106.514,E2 19106.514} C_VEL
LIN {X 0,Y 259.183,Z 648.496,A -85,B 0,C 180,E1 19109.003,E2 19109.003} C_VEL
LIN {X 0,Y 263.136,Z 642.512,A -85,B 0,C 180,E1 19109.652,E2 19109.652} C_VEL
LIN {X 0,Y 268.4,Z 660.954,A -85,B 0,C 180,E1 19115.593,E2 19115.593} C_VEL
LIN {X 0,Y 270.633,Z 676.795,A -85,B 0,C 180,E1 19119.772,E2 19119.772} C_VEL
LIN {X 0,Y 257.206,Z 708.941,A -85,B 0,C 180,E1 19124.047,E2 19124.047} C_VEL
LIN {X 0,Y 243.433,Z 735.911,A -85,B 0,C 180,E1 19129.387,E2 19129.387} C_VEL
LIN {X 0,Y 229.235,Z 759.987,A -85,B 0,C 180,E1 19136.54,E2 19136.54} C_VEL
LIN {X 0,Y 218.104,Z 778.007,A -85,B 0,C 180,E1 19144.81,E2 19144.81} C_VEL
LIN {X 0,Y 210.305,Z 791.379,A -85,B 0,C 180,E1 19154.67,E2 19154.67} C_VEL
LIN {X 0,Y 207.175,Z 798.215,A -85,B 0,C 180,E1 19163.728,E2 19163.728} C_VEL
LIN {X 0,Y 206.512,Z 800.463,A -85,B 0,C 180,E1 19170.001,E2 19170.001} C_VEL
LIN {X 0,Y 206.429,Z 800.486,A -85,B 0,C 180,E1 19178.409,E2 19178.409} C_VEL
LIN {X 0,Y 208.52,Z 796.979,A -85,B 0,C 180,E1 19186.829,E2 19186.829} C_VEL
LIN {X 0,Y 214.843,Z 787.365,A -85,B 0,C 180,E1 19197.168,E2 19197.168} C_VEL
LIN {X 0,Y 224.896,Z 773.145,A -85,B 0,C 180,E1 19205.9,E2 19205.9} C_VEL
LIN {X 0,Y 237.951,Z 754.192,A -85,B 0,C 180,E1 19213.322,E2 19213.322} C_VEL
LIN {X 0,Y 253.336,Z 729.322,A -85,B 0,C 180,E1 19219.728,E2 19219.728} C_VEL
LIN {X 0,Y 268.975,Z 699.363,A -85,B 0,C 180,E1 19224.766,E2 19224.766} C_VEL
LIN {X 0,Y 269.029,Z 698.234,A -85,B 0,C 180,E1 19225.073,E2 19225.073} C_VEL
LIN {X 0,Y 246.793,Z 712.447,A -85,B 0,C 180,E1 19228.885,E2 19228.885} C_VEL
LIN {X 0,Y 222.774,Z 724.648,A -85,B 0,C 180,E1 19236.01,E2 19236.01} C_VEL
LIN {X 0,Y 210.836,Z 729.877,A -85,B 0,C 180,E1 19242.281,E2 19242.281} C_VEL
LIN {X 0,Y 209.396,Z 750.626,A -85,B 0,C 180,E1 19250.135,E2 19250.135} C_VEL
LIN {X 0,Y 210.039,Z 761.369,A -85,B 0,C 180,E1 19256.902,E2 19256.902} C_VEL
LIN {X 0,Y 212.779,Z 766.511,A -85,B 0,C 180,E1 19264.057,E2 19264.057} C_VEL
LIN {X 0,Y 215.521,Z 766.655,A -85,B 0,C 180,E1 19268.041,E2 19268.041} C_VEL
LIN {X 0,Y 221.039,Z 763.153,A -85,B 0,C 180,E1 19273.815,E2 19273.815} C_VEL
LIN {X 0,Y 228.149,Z 754.899,A -85,B 0,C 180,E1 19279.303,E2 19279.303} C_VEL
LIN {X 0,Y 236.88,Z 740.786,A -85,B 0,C 180,E1 19284.452,E2 19284.452} C_VEL
LIN {X 0,Y 242.654,Z 729.288,A -85,B 0,C 180,E1 19287.29,E2 19287.29} C_VEL
LIN {X 0,Y 261.644,Z 718.186,A -85,B 0,C 180,E1 19290.446,E2 19290.446} C_VEL
LIN {X 0,Y 273.641,Z 709.131,A -85,B 0,C 180,E1 19291.845,E2 19291.845} C_VEL
LIN {X 0,Y 258.912,Z 741.203,A -85,B 0,C 180,E1 19296.024,E2 19296.024} C_VEL
LIN {X 0,Y 242.793,Z 770.18,A -85,B 0,C 180,E1 19301.762,E2 19301.762} C_VEL
LIN {X 0,Y 227.727,Z 794.584,A -85,B 0,C 180,E1 19309.205,E2 19309.205} C_VEL
LIN {X 0,Y 215.576,Z 813.925,A -85,B 0,C 180,E1 19318.327,E2 19318.327} C_VEL
LIN {X 0,Y 208.163,Z 827.65,A -85,B 0,C 180,E1 19328.745,E2 19328.745} C_VEL
LIN {X 0,Y 205.64,Z 835.499,A -85,B 0,C 180,E1 19339.427,E2 19339.427} C_VEL
LIN {X 0,Y 206.045,Z 837.912,A -85,B 0,C 180,E1 19349.999,E2 19349.999} C_VEL
LIN {X 0,Y 205.609,Z 835.822,A -85,B 0,C 180,E1 19358.441,E2 19358.441} C_VEL
LIN {X 0,Y 207.393,Z 828.358,A -85,B 0,C 180,E1 19368.961,E2 19368.961} C_VEL
LIN {X 0,Y 213.548,Z 814.547,A -85,B 0,C 180,E1 19379.649,E2 19379.649} C_VEL
LIN {X 0,Y 224.229,Z 795.428,A -85,B 0,C 180,E1 19388.854,E2 19388.854} C_VEL
LIN {X 0,Y 238.099,Z 770.968,A -85,B 0,C 180,E1 19396.53,E2 19396.53} C_VEL
LIN {X 0,Y 251.605,Z 744.74,A -85,B 0,C 180,E1 19402.041,E2 19402.041} C_VEL
LIN {X 0,Y 247.271,Z 745.69,A -85,B 0,C 180,E1 19402.848,E2 19402.848} C_VEL
LIN {X 0,Y 233.944,Z 760.037,A -85,B 0,C 180,E1 19408.943,E2 19408.943} C_VEL
LIN {X 0,Y 225.308,Z 766.703,A -85,B 0,C 180,E1 19414.203,E2 19414.203} C_VEL
LIN {X 0,Y 218.649,Z 769.525,A -85,B 0,C 180,E1 19419.823,E2 19419.823} C_VEL
LIN {X 0,Y 215.182,Z 769.366,A -85,B 0,C 180,E1 19423.719,E2 19423.719} C_VEL
LIN {X 0,Y 211.492,Z 765.985,A -85,B 0,C 180,E1 19429.734,E2 19429.734} C_VEL
LIN {X 0,Y 209.494,Z 757.071,A -85,B 0,C 180,E1 19436.913,E2 19436.913} C_VEL
LIN {X 0,Y 209.239,Z 748.581,A -85,B 0,C 180,E1 19441.389,E2 19441.389} C_VEL
LIN {X 0,Y 205.572,Z 739.184,A -85,B 0,C 180,E1 19445.339,E2 19445.339} C_VEL
LIN {X 0,Y 202.66,Z 728.071,A -85,B 0,C 180,E1 19449.101,E2 19449.101} C_VEL
LIN {X 0,Y 204.243,Z 711.744,A -85,B 0,C 180,E1 19453.359,E2 19453.359} C_VEL
LIN {X 0,Y 207.691,Z 708.686,A -85,B 0,C 180,E1 19455.821,E2 19455.821} C_VEL
LIN {X 0,Y 223.043,Z 694.472,A -85,B 0,C 180,E1 19462.227,E2 19462.227} C_VEL
LIN {X 0,Y 233.72,Z 684.055,A -85,B 0,C 180,E1 19465.311,E2 19465.311} C_VEL
LIN {X 0,Y 245.865,Z 670.992,A -85,B 0,C 180,E1 19468.021,E2 19468.021} C_VEL
LIN {X 0,Y 259.112,Z 654.452,A -85,B 0,C 180,E1 19470.307,E2 19470.307} C_VEL
LIN {X 0,Y 260.603,Z 653.398,A -85,B 0,C 180,E1 19470.765,E2 19470.765} C_VEL
LIN {X 0,Y 264.312,Z 671.701,A -85,B 0,C 180,E1 19476.476,E2 19476.476} C_VEL
LIN {X 0,Y 264.542,Z 681.413,A -85,B 0,C 180,E1 19478.874,E2 19478.874} C_VEL
LIN {X 0,Y 250.755,Z 712.259,A -85,B 0,C 180,E1 19483.136,E2 19483.136} C_VEL
LIN {X 0,Y 235.589,Z 740.148,A -85,B 0,C 180,E1 19488.959,E2 19488.959} C_VEL
LIN {X 0,Y 221.193,Z 763.266,A -85,B 0,C 180,E1 19496.334,E2 19496.334} C_VEL
LIN {X 0,Y 209.322,Z 781.504,A -85,B 0,C 180,E1 19505.509,E2 19505.509} C_VEL
LIN {X 0,Y 202.321,Z 792.903,A -85,B 0,C 180,E1 19514.867,E2 19514.867} C_VEL
LIN {X 0,Y 199.366,Z 798.962,A -85,B 0,C 180,E1 19523.481,E2 19523.481} C_VEL
LIN {X 0,Y 198.655,Z 801.184,A -85,B 0,C 180,E1 19530.001,E2 19530.001} C_VEL
LIN {X 0,Y 198.634,Z 801.138,A -85,B 0,C 180,E1 19538.964,E2 19538.964} C_VEL
LIN {X 0,Y 201.852,Z 796.261,A -85,B 0,C 180,E1 19549.627,E2 19549.627} C_VEL
LIN {X 0,Y 209.721,Z 785.375,A -85,B 0,C 180,E1 19560.248,E2 19560.248} C_VEL
LIN {X 0,Y 222.277,Z 768.661,A -85,B 0,C 180,E1 19569.534,E2 19569.534} C_VEL
LIN {X 0,Y 237.448,Z 747.162,A -85,B 0,C 180,E1 19576.965,E2 19576.965} C_VEL
LIN {X 0,Y 253.732,Z 720.578,A -85,B 0,C 180,E1 19582.933,E2 19582.933} C_VEL
LIN {X 0,Y 259.978,Z 708.784,A -85,B 0,C 180,E1 19584.944,E2 19584.944} C_VEL
LIN {X 0,Y 239.585,Z 720.224,A -85,B 0,C 180,E1 19588.791,E2 19588.791} C_VEL
LIN {X 0,Y 217.744,Z 730.593,A -85,B 0,C 180,E1 19595.419,E2 19595.419} C_VEL
LIN {X 0,Y 202.728,Z 737.038,A -85,B 0,C 180,E1 19603.708,E2 19603.708} C_VEL
LIN {X 0,Y 202.228,Z 737.707,A -85,B 0,C 180,E1 19604.704,E2 19604.704} C_VEL
LIN {X 0,Y 201.496,Z 753.654,A -85,B 0,C 180,E1 19611.376,E2 19611.376} C_VEL
LIN {X 0,Y 202.388,Z 763.189,A -85,B 0,C 180,E1 19617.854,E2 19617.854} C_VEL
LIN {X 0,Y 205.025,Z 767.858,A -85,B 0,C 180,E1 19624.211,E2 19624.211} C_VEL
LIN {X 0,Y 207.897,Z 768.444,A -85,B 0,C 180,E1 19628.338,E2 19628.338} C_VEL
LIN {X 0,Y 213.732,Z 765.665,A -85,B 0,C 180,E1 19634.297,E2 19634.297} C_VEL
LIN {X 0,Y 222.692,Z 756.513,A -85,B 0,C 180,E1 19640.83,E2 19640.83} C_VEL
LIN {X 0,Y 232.193,Z 742.541,A -85,B 0,C 180,E1 19646.01,E2 19646.01} C_VEL
LIN {X 0,Y 235.925,Z 737.115,A -85,B 0,C 180,E1 19647.617,E2 19647.617} C_VEL
LIN {X 0,Y 257.848,Z 725.662,A -85,B 0,C 180,E1 19651.312,E2 19651.312} C_VEL
LIN {X 0,Y 263.18,Z 722.157,A -85,B 0,C 180,E1 19651.949,E2 19651.949} C_VEL
LIN {X 0,Y 247.251,Z 753.051,A -85,B 0,C 180,E1 19656.761,E2 19656.761} C_VEL
LIN {X 0,Y 230.805,Z 779.828,A -85,B 0,C 180,E1 19663.109,E2 19663.109} C_VEL
LIN {X 0,Y 216.238,Z 801.661,A -85,B 0,C 180,E1 19671.087,E2 19671.087} C_VEL
LIN {X 0,Y 204.927,Z 819.052,A -85,B 0,C 180,E1 19681.088,E2 19681.088} C_VEL
LIN {X 0,Y 198.957,Z 830.759,A -85,B 0,C 180,E1 19692.336,E2 19692.336} C_VEL
LIN {X 0,Y 197.675,Z 835.716,A -85,B 0,C 180,E1 19701.216,E2 19701.216} C_VEL
LIN {X 0,Y 198.178,Z 837.202,A -85,B 0,C 180,E1 19709.999,E2 19709.999} C_VEL
LIN {X 0,Y 197.729,Z 835.075,A -85,B 0,C 180,E1 19718.78,E2 19718.78} C_VEL
LIN {X 0,Y 199.711,Z 827.547,A -85,B 0,C 180,E1 19729.72,E2 19729.72} C_VEL
LIN {X 0,Y 205.589,Z 815.121,A -85,B 0,C 180,E1 19739.826,E2 19739.826} C_VEL
LIN {X 0,Y 215.965,Z 797.504,A -85,B 0,C 180,E1 19748.97,E2 19748.97} C_VEL
LIN {X 0,Y 230.017,Z 774.137,A -85,B 0,C 180,E1 19756.88,E2 19756.88} C_VEL
LIN {X 0,Y 242.027,Z 751.669,A -85,B 0,C 180,E1 19762.132,E2 19762.132} C_VEL
LIN {X 0,Y 238.288,Z 753.869,A -85,B 0,C 180,E1 19763.274,E2 19763.274} C_VEL
LIN {X 0,Y 224.481,Z 765.675,A -85,B 0,C 180,E1 19769.734,E2 19769.734} C_VEL
LIN {X 0,Y 215.888,Z 770.423,A -85,B 0,C 180,E1 19775.335,E2 19775.335} C_VEL
LIN {X 0,Y 207.769,Z 771.019,A -85,B 0,C 180,E1 19783.121,E2 19783.121} C_VEL
LIN {X 0,Y 203.326,Z 766.153,A -85,B 0,C 180,E1 19790.397,E2 19790.397} C_VEL
LIN {X 0,Y 201.508,Z 755.898,A -85,B 0,C 180,E1 19797.864,E2 19797.864} C_VEL
LIN {X 0,Y 201.695,Z 740.788,A -85,B 0,C 180,E1 19804.838,E2 19804.838} C_VEL
LIN {X 0,Y 202.66,Z 728.071,A -85,B 0,C 180,E1 19809.101,E2 19809.101} C_VEL
LIN {X 0,Y 202.428,Z 721.161,A -85,B 0,C 180,E1 19812.262,E2 19812.262} C_VEL
LIN {X 0,Y 204.481,Z 714.087,A -85,B 0,C 180,E1 19817.047,E2 19817.047} C_VEL
LIN {X 0,Y 205.924,Z 712.609,A -85,B 0,C 180,E1 19817.742,E2 19817.742} C_VEL
LIN {X 0,Y 219.647,Z 701.03,A -85,B 0,C 180,E1 19823.278,E2 19823.278} C_VEL
LIN {X 0,Y 240.616,Z 681.399,A -85,B 0,C 180,E1 19828.587,E2 19828.587} C_VEL
LIN {X 0,Y 257.058,Z 662.992,A -85,B 0,C 180,E1 19831.408,E2 19831.408} C_VEL
LIN {X 0,Y 259.48,Z 681.767,A -85,B 0,C 180,E1 19837.197,E2 19837.197} C_VEL
LIN {X 0,Y 257.311,Z 688.407,A -85,B 0,C 180,E1 19838.187,E2 19838.187} C_VEL
LIN {X 0,Y 242.504,Z 719.005,A -85,B 0,C 180,E1 19842.777,E2 19842.777} C_VEL
LIN {X 0,Y 226.841,Z 745.836,A -85,B 0,C 180,E1 19848.93,E2 19848.93} C_VEL
LIN {X 0,Y 212.415,Z 767.548,A -85,B 0,C 180,E1 19856.591,E2 19856.591} C_VEL
LIN {X 0,Y 201.126,Z 783.837,A -85,B 0,C 180,E1 19865.626,E2 19865.626} C_VEL
LIN {X 0,Y 193.658,Z 795.548,A -85,B 0,C 180,E1 19876.481,E2 19876.481} C_VEL
LIN {X 0,Y 191.178,Z 800.67,A -85,B 0,C 180,E1 19885.473,E2 19885.473} C_VEL
LIN {X 0,Y 190.497,Z 802.358,A -85,B 0,C 180,E1 19894.545,E2 19894.545} C_VEL
LIN {X 0,Y 192.406,Z 799.577,A -85,B 0,C 180,E1 19905.935,E2 19905.935} C_VEL
LIN {X 0,Y 198.799,Z 791.109,A -85,B 0,C 180,E1 19917.097,E2 19917.097} C_VEL
LIN {X 0,Y 209.974,Z 777.134,A -85,B 0,C 180,E1 19927.041,E2 19927.041} C_VEL
LIN {X 0,Y 224.978,Z 757.716,A -85,B 0,C 180,E1 19935.378,E2 19935.378} C_VEL
LIN {X 0,Y 241.851,Z 733.012,A -85,B 0,C 180,E1 19942.085,E2 19942.085} C_VEL
LIN {X 0,Y 249.92,Z 718.894,A -85,B 0,C 180,E1 19944.994,E2 19944.994} C_VEL
LIN {X 0,Y 225.817,Z 730.688,A -85,B 0,C 180,E1 19950.323,E2 19950.323} C_VEL
LIN {X 0,Y 204.759,Z 739.625,A -85,B 0,C 180,E1 19958.367,E2 19958.367} C_VEL
LIN {X 0,Y 193.94,Z 744.06,A -85,B 0,C 180,E1 19966.777,E2 19966.777} C_VEL
LIN {X 0,Y 193.72,Z 757.528,A -85,B 0,C 180,E1 19973.28,E2 19973.28} C_VEL
LIN {X 0,Y 195.202,Z 766.041,A -85,B 0,C 180,E1 19979.99,E2 19979.99} C_VEL
LIN {X 0,Y 197.233,Z 769.078,A -85,B 0,C 180,E1 19984.378,E2 19984.378} C_VEL
LIN {X 0,Y 200.251,Z 770.127,A -85,B 0,C 180,E1 19988.658,E2 19988.658} C_VEL
LIN {X 0,Y 206.404,Z 768.055,A -85,B 0,C 180,E1 19994.816,E2 19994.816} C_VEL
LIN {X 0,Y 215.894,Z 759.904,A -85,B 0,C 180,E1 20001.518,E2 20001.518} C_VEL
LIN {X 0,Y 226.841,Z 745.86,A -85,B 0,C 180,E1 20007.206,E2 20007.206} C_VEL
LIN {X 0,Y 247.063,Z 736.44,A -85,B 0,C 180,E1 20011.218,E2 20011.218} C_VEL
LIN {X 0,Y 252.806,Z 733.344,A -85,B 0,C 180,E1 20012.028,E2 20012.028} C_VEL
LIN {X 0,Y 235.559,Z 763.307,A -85,B 0,C 180,E1 20017.499,E2 20017.499} C_VEL
LIN {X 0,Y 218.789,Z 788.302,A -85,B 0,C 180,E1 20024.556,E2 20024.556} C_VEL
LIN {X 0,Y 204.172,Z 808.876,A -85,B 0,C 180,E1 20033.747,E2 20033.747} C_VEL
LIN {X 0,Y 194.345,Z 823.938,A -85,B 0,C 180,E1 20044.715,E2 20044.715} C_VEL
LIN {X 0,Y 190.222,Z 832.952,A -85,B 0,C 180,E1 20056.23,E2 20056.23} C_VEL
LIN {X 0,Y 189.704,Z 836.167,A -85,B 0,C 180,E1 20065.436,E2 20065.436} C_VEL
LIN {X 0,Y 190.308,Z 836.492,A -85,B 0,C 180,E1 20069.999,E2 20069.999} C_VEL
LIN {X 0,Y 189.847,Z 834.331,A -85,B 0,C 180,E1 20079.147,E2 20079.147} C_VEL
LIN {X 0,Y 191.58,Z 828.024,A -85,B 0,C 180,E1 20089.086,E2 20089.086} C_VEL
LIN {X 0,Y 197.455,Z 816.023,A -85,B 0,C 180,E1 20099.788,E2 20099.788} C_VEL
LIN {X 0,Y 208.847,Z 797.65,A -85,B 0,C 180,E1 20109.89,E2 20109.89} C_VEL
LIN {X 0,Y 223.453,Z 774.555,A -85,B 0,C 180,E1 20117.981,E2 20117.981} C_VEL
LIN {X 0,Y 232.991,Z 757.853,A -85,B 0,C 180,E1 20122.219,E2 20122.219} C_VEL
LIN {X 0,Y 218.196,Z 768.657,A -85,B 0,C 180,E1 20128.766,E2 20128.766} C_VEL
LIN {X 0,Y 209.171,Z 772.682,A -85,B 0,C 180,E1 20134.361,E2 20134.361} C_VEL
LIN {X 0,Y 204.327,Z 773.43,A -85,B 0,C 180,E1 20138.34,E2 20138.34} C_VEL
LIN {X 0,Y 197.303,Z 770.113,A -85,B 0,C 180,E1 20146.746,E2 20146.746} C_VEL
LIN {X 0,Y 194.143,Z 761.739,A -85,B 0,C 180,E1 20154.435,E2 20154.435} C_VEL
LIN {X 0,Y 193.515,Z 747.453,A -85,B 0,C 180,E1 20162.245,E2 20162.245} C_VEL
LIN {X 0,Y 194.859,Z 727.482,A -85,B 0,C 180,E1 20169.482,E2 20169.482} C_VEL
LIN {X 0,Y 195.374,Z 722.179,A -85,B 0,C 180,E1 20171.144,E2 20171.144} C_VEL
LIN {X 0,Y 204.481,Z 713.959,A -85,B 0,C 180,E1 20177.179,E2 20177.179} C_VEL
LIN {X 0,Y 205.924,Z 712.609,A -85,B 0,C 180,E1 20177.742,E2 20177.742} C_VEL
LIN {X 0,Y 211.571,Z 708.515,A -85,B 0,C 180,E1 20180.735,E2 20180.735} C_VEL
LIN {X 0,Y 220.013,Z 703.872,A -85,B 0,C 180,E1 20185.28,E2 20185.28} C_VEL
LIN {X 0,Y 221.222,Z 702.946,A -85,B 0,C 180,E1 20185.683,E2 20185.683} C_VEL
LIN {X 0,Y 239.315,Z 687.012,A -85,B 0,C 180,E1 20189.915,E2 20189.915} C_VEL
LIN {X 0,Y 250.727,Z 674.89,A -85,B 0,C 180,E1 20191.707,E2 20191.707} C_VEL
LIN {X 0,Y 253.185,Z 673.544,A -85,B 0,C 180,E1 20192.449,E2 20192.449} C_VEL
LIN {X 0,Y 254.082,Z 685.351,A -85,B 0,C 180,E1 20196.124,E2 20196.124} C_VEL
LIN {X 0,Y 239.794,Z 715.644,A -85,B 0,C 180,E1 20200.61,E2 20200.61} C_VEL
LIN {X 0,Y 224.011,Z 742.199,A -85,B 0,C 180,E1 20206.327,E2 20206.327} C_VEL
LIN {X 0,Y 208.203,Z 765.209,A -85,B 0,C 180,E1 20213.969,E2 20213.969} C_VEL
LIN {X 0,Y 195.087,Z 783.199,A -85,B 0,C 180,E1 20223.589,E2 20223.589} C_VEL
LIN {X 0,Y 187.151,Z 794.481,A -85,B 0,C 180,E1 20233.607,E2 20233.607} C_VEL
LIN {X 0,Y 183.349,Z 801.404,A -85,B 0,C 180,E1 20245.279,E2 20245.279} C_VEL
LIN {X 0,Y 182.639,Z 803.061,A -85,B 0,C 180,E1 20254.741,E2 20254.741} C_VEL
LIN {X 0,Y 184.773,Z 800.267,A -85,B 0,C 180,E1 20266.612,E2 20266.612} C_VEL
LIN {X 0,Y 191.686,Z 791.782,A -85,B 0,C 180,E1 20278.191,E2 20278.191} C_VEL
LIN {X 0,Y 203.29,Z 778.184,A -85,B 0,C 180,E1 20288.192,E2 20288.192} C_VEL
LIN {X 0,Y 218.308,Z 759.812,A -85,B 0,C 180,E1 20296.365,E2 20296.365} C_VEL
LIN {X 0,Y 235.7,Z 735.639,A -85,B 0,C 180,E1 20303.167,E2 20303.167} C_VEL
LIN {X 0,Y 240.436,Z 728.395,A -85,B 0,C 180,E1 20304.686,E2 20304.686} C_VEL
LIN {X 0,Y 233.671,Z 730.895,A -85,B 0,C 180,E1 20306.34,E2 20306.34} C_VEL
LIN {X 0,Y 207.3,Z 741.988,A -85,B 0,C 180,E1 20314.092,E2 20314.092} C_VEL
LIN {X 0,Y 192.892,Z 747.551,A -85,B 0,C 180,E1 20321.753,E2 20321.753} C_VEL
LIN {X 0,Y 185.824,Z 750.526,A -85,B 0,C 180,E1 20329.345,E2 20329.345} C_VEL
LIN {X 0,Y 186.341,Z 762.752,A -85,B 0,C 180,E1 20336.507,E2 20336.507} C_VEL
LIN {X 0,Y 189.429,Z 770.229,A -85,B 0,C 180,E1 20344.559,E2 20344.559} C_VEL
LIN {X 0,Y 192.588,Z 771.73,A -85,B 0,C 180,E1 20349.006,E2 20349.006} C_VEL
LIN {X 0,Y 199.098,Z 770.408,A -85,B 0,C 180,E1 20355.373,E2 20355.373} C_VEL
LIN {X 0,Y 209.137,Z 763.297,A -85,B 0,C 180,E1 20362.25,E2 20362.25} C_VEL
LIN {X 0,Y 219.746,Z 751.77,A -85,B 0,C 180,E1 20367.605,E2 20367.605} C_VEL
LIN {X 0,Y 238.423,Z 745.007,A -85,B 0,C 180,E1 20371.442,E2 20371.442} C_VEL
LIN {X 0,Y 241.856,Z 743.465,A -85,B 0,C 180,E1 20371.969,E2 20371.969} C_VEL
LIN {X 0,Y 237.538,Z 751.701,A -85,B 0,C 180,E1 20373.647,E2 20373.647} C_VEL
LIN {X 0,Y 219.472,Z 778.697,A -85,B 0,C 180,E1 20380.092,E2 20380.092} C_VEL
LIN {X 0,Y 202.853,Z 801.198,A -85,B 0,C 180,E1 20388.678,E2 20388.678} C_VEL
LIN {X 0,Y 190.45,Z 817.967,A -85,B 0,C 180,E1 20398.996,E2 20398.996} C_VEL
LIN {X 0,Y 183.576,Z 829.343,A -85,B 0,C 180,E1 20410.801,E2 20410.801} C_VEL
LIN {X 0,Y 181.939,Z 834.303,A -85,B 0,C 180,E1 20420.45,E2 20420.45} C_VEL
LIN {X 0,Y 182.438,Z 835.782,A -85,B 0,C 180,E1 20429.999,E2 20429.999} C_VEL
LIN {X 0,Y 181.982,Z 833.583,A -85,B 0,C 180,E1 20439.546,E2 20439.546} C_VEL
LIN {X 0,Y 183.905,Z 827.217,A -85,B 0,C 180,E1 20449.916,E2 20449.916} C_VEL
LIN {X 0,Y 190.364,Z 815.13,A -85,B 0,C 180,E1 20461.017,E2 20461.017} C_VEL
LIN {X 0,Y 202.567,Z 796.655,A -85,B 0,C 180,E1 20471.391,E2 20471.391} C_VEL
LIN {X 0,Y 217.96,Z 773.446,A -85,B 0,C 180,E1 20479.609,E2 20479.609} C_VEL
LIN {X 0,Y 223.882,Z 764.588,A -85,B 0,C 180,E1 20482.041,E2 20482.041} C_VEL
LIN {X 0,Y 221.567,Z 766.116,A -85,B 0,C 180,E1 20483.432,E2 20483.432} C_VEL
LIN {X 0,Y 208.56,Z 773.091,A -85,B 0,C 180,E1 20489.581,E2 20489.581} C_VEL
LIN {X 0,Y 197.217,Z 775.272,A -85,B 0,C 180,E1 20497.517,E2 20497.517} C_VEL
LIN {X 0,Y 191.181,Z 772.921,A -85,B 0,C 180,E1 20503.974,E2 20503.974} C_VEL
LIN {X 0,Y 187,Z 765.446,A -85,B 0,C 180,E1 20511.892,E2 20511.892} C_VEL
LIN {X 0,Y 185.623,Z 751.235,A -85,B 0,C 180,E1 20520.593,E2 20520.593} C_VEL
LIN {X 0,Y 186.724,Z 731.824,A -85,B 0,C 180,E1 20528.726,E2 20528.726} C_VEL
LIN {X 0,Y 199.151,Z 720.895,A -85,B 0,C 180,E1 20537.654,E2 20537.654} C_VEL
LIN {X 0,Y 219.178,Z 704.808,A -85,B 0,C 180,E1 20545.163,E2 20545.163} C_VEL
LIN {X 0,Y 221.222,Z 702.946,A -85,B 0,C 180,E1 20545.683,E2 20545.683} C_VEL
LIN {X 0,Y 238.766,Z 691.687,A -85,B 0,C 180,E1 20551.322,E2 20551.322} C_VEL
LIN {X 0,Y 241.536,Z 689.262,A -85,B 0,C 180,E1 20551.867,E2 20551.867} C_VEL
LIN {X 0,Y 247.561,Z 683.141,A -85,B 0,C 180,E1 20552.719,E2 20552.719} C_VEL
LIN {X 0,Y 248.549,Z 683.019,A -85,B 0,C 180,E1 20553.131,E2 20553.131} C_VEL
LIN {X 0,Y 248.404,Z 690.093,A -85,B 0,C 180,E1 20555.25,E2 20555.25} C_VEL
LIN {X 0,Y 233.052,Z 719.834,A -85,B 0,C 180,E1 20559.682,E2 20559.682} C_VEL
LIN {X 0,Y 216.271,Z 746.343,A -85,B 0,C 180,E1 20565.749,E2 20565.749} C_VEL
LIN {X 0,Y 200.27,Z 768.265,A -85,B 0,C 180,E1 20573.6,E2 20573.6} C_VEL
LIN {X 0,Y 186.882,Z 785.514,A -85,B 0,C 180,E1 20583.632,E2 20583.632} C_VEL
LIN {X 0,Y 178.375,Z 797.1,A -85,B 0,C 180,E1 20595.297,E2 20595.297} C_VEL
LIN {X 0,Y 175.519,Z 802.138,A -85,B 0,C 180,E1 20605.068,E2 20605.068} C_VEL
LIN {X 0,Y 174.773,Z 803.765,A -85,B 0,C 180,E1 20614.955,E2 20614.955} C_VEL
LIN {X 0,Y 177.152,Z 800.956,A -85,B 0,C 180,E1 20627.349,E2 20627.349} C_VEL
LIN {X 0,Y 184.638,Z 792.466,A -85,B 0,C 180,E1 20639.369,E2 20639.369} C_VEL
LIN {X 0,Y 196.619,Z 779.317,A -85,B 0,C 180,E1 20649.37,E2 20649.37} C_VEL
LIN {X 0,Y 213.55,Z 759.636,A -85,B 0,C 180,E1 20658.222,E2 20658.222} C_VEL
LIN {X 0,Y 229.798,Z 738.054,A -85,B 0,C 180,E1 20664.345,E2 20664.345} C_VEL
LIN {X 0,Y 230.532,Z 736.09,A -85,B 0,C 180,E1 20665.074,E2 20665.074} C_VEL
LIN {X 0,Y 204.557,Z 746.429,A -85,B 0,C 180,E1 20672.295,E2 20672.295} C_VEL
LIN {X 0,Y 187.237,Z 752.761,A -85,B 0,C 180,E1 20681.182,E2 20681.182} C_VEL
LIN {X 0,Y 177.907,Z 757.269,A -85,B 0,C 180,E1 20692.679,E2 20692.679} C_VEL
LIN {X 0,Y 179.886,Z 768.435,A -85,B 0,C 180,E1 20701.191,E2 20701.191} C_VEL
LIN {X 0,Y 184.924,Z 773.241,A -85,B 0,C 180,E1 20709.382,E2 20709.382} C_VEL
LIN {X 0,Y 189.198,Z 773.335,A -85,B 0,C 180,E1 20713.833,E2 20713.833} C_VEL
LIN {X 0,Y 199.098,Z 768.921,A -85,B 0,C 180,E1 20721.091,E2 20721.091} C_VEL
LIN {X 0,Y 211.558,Z 758.336,A -85,B 0,C 180,E1 20727.612,E2 20727.612} C_VEL
LIN {X 0,Y 232.047,Z 752.488,A -85,B 0,C 180,E1 20732.274,E2 20732.274} C_VEL
LIN {X 0,Y 213.164,Z 779.363,A -85,B 0,C 180,E1 20738.849,E2 20738.849} C_VEL
LIN {X 0,Y 195.9,Z 801.521,A -85,B 0,C 180,E1 20747.616,E2 20747.616} C_VEL
LIN {X 0,Y 182.42,Z 818.638,A -85,B 0,C 180,E1 20758.863,E2 20758.863} C_VEL
LIN {X 0,Y 175.632,Z 829.239,A -85,B 0,C 180,E1 20770.896,E2 20770.896} C_VEL
LIN {X 0,Y 174.066,Z 833.594,A -85,B 0,C 180,E1 20780.013,E2 20780.013} C_VEL
LIN {X 0,Y 174.543,Z 835.07,A -85,B 0,C 180,E1 20789.999,E2 20789.999} C_VEL
LIN {X 0,Y 174.109,Z 832.836,A -85,B 0,C 180,E1 20799.982,E2 20799.982} C_VEL
LIN {X 0,Y 176.478,Z 825.994,A -85,B 0,C 180,E1 20811.311,E2 20811.311} C_VEL
LIN {X 0,Y 184.428,Z 812.579,A -85,B 0,C 180,E1 20823.528,E2 20823.528} C_VEL
LIN {X 0,Y 198.017,Z 793.497,A -85,B 0,C 180,E1 20833.949,E2 20833.949} C_VEL
LIN {X 0,Y 214.144,Z 770.862,A -85,B 0,C 180,E1 20841.892,E2 20841.892} C_VEL
LIN {X 0,Y 214.72,Z 770.351,A -85,B 0,C 180,E1 20842.782,E2 20842.782} C_VEL
LIN {X 0,Y 202.181,Z 775.734,A -85,B 0,C 180,E1 20848.514,E2 20848.514} C_VEL
LIN {X 0,Y 190.123,Z 777.119,A -85,B 0,C 180,E1 20856.63,E2 20856.63} C_VEL
LIN {X 0,Y 182.065,Z 772.377,A -85,B 0,C 180,E1 20865.613,E2 20865.613} C_VEL
LIN {X 0,Y 178.462,Z 762.839,A -85,B 0,C 180,E1 20873.944,E2 20873.944} C_VEL
LIN {X 0,Y 177.757,Z 747.333,A -85,B 0,C 180,E1 20882.444,E2 20882.444} C_VEL
LIN {X 0,Y 178.157,Z 741.061,A -85,B 0,C 180,E1 20885.479,E2 20885.479} C_VEL
LIN {X 0,Y 189.601,Z 730.567,A -85,B 0,C 180,E1 20895.782,E2 20895.782} C_VEL
LIN {X 0,Y 207.682,Z 716.967,A -85,B 0,C 180,E1 20903.759,E2 20903.759} C_VEL
LIN {X 0,Y 227.163,Z 701.939,A -85,B 0,C 180,E1 20909.133,E2 20909.133} C_VEL
LIN {X 0,Y 241.536,Z 689.262,A -85,B 0,C 180,E1 20911.867,E2 20911.867} C_VEL
LIN {X 0,Y 243.066,Z 689.813,A -85,B 0,C 180,E1 20912.777,E2 20912.777} C_VEL
LIN {X 0,Y 241.265,Z 696.785,A -85,B 0,C 180,E1 20914.376,E2 20914.376} C_VEL
LIN {X 0,Y 231.644,Z 715.005,A -85,B 0,C 180,E1 20917.141,E2 20917.141} C_VEL
LIN {X 0,Y 214.069,Z 742.708,A -85,B 0,C 180,E1 20922.994,E2 20922.994} C_VEL
LIN {X 0,Y 197.369,Z 764.947,A -85,B 0,C 180,E1 20930.337,E2 20930.337} C_VEL
LIN {X 0,Y 182.4,Z 783.303,A -85,B 0,C 180,E1 20940.236,E2 20940.236} C_VEL
LIN {X 0,Y 172.06,Z 796.057,A -85,B 0,C 180,E1 20952.123,E2 20952.123} C_VEL
LIN {X 0,Y 167.694,Z 802.87,A -85,B 0,C 180,E1 20964.838,E2 20964.838} C_VEL
LIN {X 0,Y 166.882,Z 804.444,A -85,B 0,C 180,E1 20975.802,E2 20975.802} C_VEL
LIN {X 0,Y 169.563,Z 801.648,A -85,B 0,C 180,E1 20988.151,E2 20988.151} C_VEL
LIN {X 0,Y 177.693,Z 793.137,A -85,B 0,C 180,E1 21000.638,E2 21000.638} C_VEL
LIN {X 0,Y 190.481,Z 779.986,A -85,B 0,C 180,E1 21010.902,E2 21010.902} C_VEL
LIN {X 0,Y 208.197,Z 760.427,A -85,B 0,C 180,E1 21019.814,E2 21019.814} C_VEL
LIN {X 0,Y 221.632,Z 743.66,A -85,B 0,C 180,E1 21024.799,E2 21024.799} C_VEL
LIN {X 0,Y 192.041,Z 754.135,A -85,B 0,C 180,E1 21034.383,E2 21034.383} C_VEL
LIN {X 0,Y 176.421,Z 759.54,A -85,B 0,C 180,E1 21045.12,E2 21045.12} C_VEL
LIN {X 0,Y 170.502,Z 762.898,A -85,B 0,C 180,E1 21056.182,E2 21056.182} C_VEL
LIN {X 0,Y 173.784,Z 772.106,A -85,B 0,C 180,E1 21064.97,E2 21064.97} C_VEL
LIN {X 0,Y 177.231,Z 774.603,A -85,B 0,C 180,E1 21069.793,E2 21069.793} C_VEL
LIN {X 0,Y 181.755,Z 775.222,A -85,B 0,C 180,E1 21074.412,E2 21074.412} C_VEL
LIN {X 0,Y 190.517,Z 772.629,A -85,B 0,C 180,E1 21080.87,E2 21080.87} C_VEL
LIN {X 0,Y 203.521,Z 764.392,A -85,B 0,C 180,E1 21087.69,E2 21087.69} C_VEL
LIN {X 0,Y 222.151,Z 759.651,A -85,B 0,C 180,E1 21092.116,E2 21092.116} C_VEL
LIN {X 0,Y 202.752,Z 785.313,A -85,B 0,C 180,E1 21099.319,E2 21099.319} C_VEL
LIN {X 0,Y 186.27,Z 804.981,A -85,B 0,C 180,E1 21108.227,E2 21108.227} C_VEL
LIN {X 0,Y 173.38,Z 820.542,A -85,B 0,C 180,E1 21119.95,E2 21119.95} C_VEL
LIN {X 0,Y 167.294,Z 829.894,A -85,B 0,C 180,E1 21132.343,E2 21132.343} C_VEL
LIN {X 0,Y 166.213,Z 832.889,A -85,B 0,C 180,E1 21139.536,E2 21139.536} C_VEL
LIN {X 0,Y 166.671,Z 834.359,A -85,B 0,C 180,E1 21149.999,E2 21149.999} C_VEL
LIN {X 0,Y 166.268,Z 832.09,A -85,B 0,C 180,E1 21160.458,E2 21160.458} C_VEL
LIN {X 0,Y 168.92,Z 825.18,A -85,B 0,C 180,E1 21172.315,E2 21172.315} C_VEL
LIN {X 0,Y 177.63,Z 811.688,A -85,B 0,C 180,E1 21184.993,E2 21184.993} C_VEL
LIN {X 0,Y 192.261,Z 792.303,A -85,B 0,C 180,E1 21195.747,E2 21195.747} C_VEL
LIN {X 0,Y 204.68,Z 776.079,A -85,B 0,C 180,E1 21201.843,E2 21201.843} C_VEL
LIN {X 0,Y 205.764,Z 775.22,A -85,B 0,C 180,E1 21202.913,E2 21202.913} C_VEL
LIN {X 0,Y 195.878,Z 778.356,A -85,B 0,C 180,E1 21207.378,E2 21207.378} C_VEL
LIN {X 0,Y 183.057,Z 778.827,A -85,B 0,C 180,E1 21215.67,E2 21215.67} C_VEL
LIN {X 0,Y 174.489,Z 773.399,A -85,B 0,C 180,E1 21224.974,E2 21224.974} C_VEL
LIN {X 0,Y 170.611,Z 763.199,A -85,B 0,C 180,E1 21233.664,E2 21233.664} C_VEL
LIN {X 0,Y 169.883,Z 750.133,A -85,B 0,C 180,E1 21241.284,E2 21241.284} C_VEL
LIN {X 0,Y 180.29,Z 739.473,A -85,B 0,C 180,E1 21253.693,E2 21253.693} C_VEL
LIN {X 0,Y 199.114,Z 726.166,A -85,B 0,C 180,E1 21263.359,E2 21263.359} C_VEL
LIN {X 0,Y 221.198,Z 710.368,A -85,B 0,C 180,E1 21269.655,E2 21269.655} C_VEL
LIN {X 0,Y 240.186,Z 694.861,A -85,B 0,C 180,E1 21273.22,E2 21273.22} C_VEL
LIN {X 0,Y 243.254,Z 692.912,A -85,B 0,C 180,E1 21273.949,E2 21273.949} C_VEL
LIN {X 0,Y 231.644,Z 715.005,A -85,B 0,C 180,E1 21277.141,E2 21277.141} C_VEL
LIN {X 0,Y 221.561,Z 728.17,A -85,B 0,C 180,E1 21278.679,E2 21278.679} C_VEL
LIN {X 0,Y 212.3,Z 738.864,A -85,B 0,C 180,E1 21280.194,E2 21280.194} C_VEL
LIN {X 0,Y 211.259,Z 740.283,A -85,B 0,C 180,E1 21280.535,E2 21280.535} C_VEL
LIN {X 0,Y 192.955,Z 763.954,A -85,B 0,C 180,E1 21288.044,E2 21288.044} C_VEL
LIN {X 0,Y 177.076,Z 782.513,A -85,B 0,C 180,E1 21297.815,E2 21297.815} C_VEL
LIN {X 0,Y 165.38,Z 795.88,A -85,B 0,C 180,E1 21309.99,E2 21309.99} C_VEL
LIN {X 0,Y 160.158,Z 802.956,A -85,B 0,C 180,E1 21322.573,E2 21322.573} C_VEL
LIN {X 0,Y 159.306,Z 804.79,A -85,B 0,C 180,E1 21330.001,E2 21330.001} C_VEL
LIN {X 0,Y 159.569,Z 804.676,A -85,B 0,C 180,E1 21340.905,E2 21340.905} C_VEL
LIN {X 0,Y 163.911,Z 800.471,A -85,B 0,C 180,E1 21352.95,E2 21352.95} C_VEL
LIN {X 0,Y 174.789,Z 790.068,A -85,B 0,C 180,E1 21365.674,E2 21365.674} C_VEL
LIN {X 0,Y 191.025,Z 774.065,A -85,B 0,C 180,E1 21376.131,E2 21376.131} C_VEL
LIN {X 0,Y 209.996,Z 753.09,A -85,B 0,C 180,E1 21384.128,E2 21384.128} C_VEL
LIN {X 0,Y 211.406,Z 750.655,A -85,B 0,C 180,E1 21385.165,E2 21385.165} C_VEL
LIN {X 0,Y 185.935,Z 759.228,A -85,B 0,C 180,E1 21393.736,E2 21393.736} C_VEL
LIN {X 0,Y 166.338,Z 766.11,A -85,B 0,C 180,E1 21409.534,E2 21409.534} C_VEL
LIN {X 0,Y 164.064,Z 769.305,A -85,B 0,C 180,E1 21421.306,E2 21421.306} C_VEL
LIN {X 0,Y 169.555,Z 775.847,A -85,B 0,C 180,E1 21430.241,E2 21430.241} C_VEL
LIN {X 0,Y 174.282,Z 776.981,A -85,B 0,C 180,E1 21435.044,E2 21435.044} C_VEL
LIN {X 0,Y 183.52,Z 775.243,A -85,B 0,C 180,E1 21441.705,E2 21441.705} C_VEL
LIN {X 0,Y 195.108,Z 770.048,A -85,B 0,C 180,E1 21447.638,E2 21447.638} C_VEL
LIN {X 0,Y 211.987,Z 766.853,A -85,B 0,C 180,E1 21452.191,E2 21452.191} C_VEL
LIN {X 0,Y 192.001,Z 791.02,A -85,B 0,C 180,E1 21459.969,E2 21459.969} C_VEL
LIN {X 0,Y 175.583,Z 809.234,A -85,B 0,C 180,E1 21469.657,E2 21469.657} C_VEL
LIN {X 0,Y 163.515,Z 823.323,A -85,B 0,C 180,E1 21482.516,E2 21482.516} C_VEL
LIN {X 0,Y 158.63,Z 831.256,A -85,B 0,C 180,E1 21496.24,E2 21496.24} C_VEL
LIN {X 0,Y 158.129,Z 833.355,A -85,B 0,C 180,E1 21504.522,E2 21504.522} C_VEL
LIN {X 0,Y 158.794,Z 833.648,A -85,B 0,C 180,E1 21509.999,E2 21509.999} C_VEL
LIN {X 0,Y 158.403,Z 831.338,A -85,B 0,C 180,E1 21520.984,E2 21520.984} C_VEL
LIN {X 0,Y 161.41,Z 824.37,A -85,B 0,C 180,E1 21533.413,E2 21533.413} C_VEL
LIN {X 0,Y 170.97,Z 810.779,A -85,B 0,C 180,E1 21546.571,E2 21546.571} C_VEL
LIN {X 0,Y 186.551,Z 791.283,A -85,B 0,C 180,E1 21557.577,E2 21557.577} C_VEL
LIN {X 0,Y 195.153,Z 780.438,A -85,B 0,C 180,E1 21561.799,E2 21561.799} C_VEL
LIN {X 0,Y 196.932,Z 779.272,A -85,B 0,C 180,E1 21562.896,E2 21562.896} C_VEL
LIN {X 0,Y 182.295,Z 781.368,A -85,B 0,C 180,E1 21570.232,E2 21570.232} C_VEL
LIN {X 0,Y 170.887,Z 778.147,A -85,B 0,C 180,E1 21579.328,E2 21579.328} C_VEL
LIN {X 0,Y 164.096,Z 768.757,A -85,B 0,C 180,E1 21589.414,E2 21589.414} C_VEL
LIN {X 0,Y 162.218,Z 758.872,A -85,B 0,C 180,E1 21596.679,E2 21596.679} C_VEL
LIN {X 0,Y 175.604,Z 744.477,A -85,B 0,C 180,E1 21614.951,E2 21614.951} C_VEL
LIN {X 0,Y 195.949,Z 731.14,A -85,B 0,C 180,E1 21624.871,E2 21624.871} C_VEL
LIN {X 0,Y 219.077,Z 715.523,A -85,B 0,C 180,E1 21631.116,E2 21631.116} C_VEL
LIN {X 0,Y 232.453,Z 705.339,A -85,B 0,C 180,E1 21633.529,E2 21633.529} C_VEL
LIN {X 0,Y 231.326,Z 708.693,A -85,B 0,C 180,E1 21634.377,E2 21634.377} C_VEL
LIN {X 0,Y 213.726,Z 736.771,A -85,B 0,C 180,E1 21639.653,E2 21639.653} C_VEL
LIN {X 0,Y 211.259,Z 740.283,A -85,B 0,C 180,E1 21640.535,E2 21640.535} C_VEL
LIN {X 0,Y 200.581,Z 751.687,A -85,B 0,C 180,E1 21642.766,E2 21642.766} C_VEL
LIN {X 0,Y 189.619,Z 762.173,A -85,B 0,C 180,E1 21645.338,E2 21645.338} C_VEL
LIN {X 0,Y 172.034,Z 781.725,A -85,B 0,C 180,E1 21655.236,E2 21655.236} C_VEL
LIN {X 0,Y 158.943,Z 795.634,A -85,B 0,C 180,E1 21667.68,E2 21667.68} C_VEL
LIN {X 0,Y 153.329,Z 802.342,A -85,B 0,C 180,E1 21678.648,E2 21678.648} C_VEL
LIN {X 0,Y 151.445,Z 805.512,A -85,B 0,C 180,E1 21690.001,E2 21690.001} C_VEL
LIN {X 0,Y 151.792,Z 805.375,A -85,B 0,C 180,E1 21701.471,E2 21701.471} C_VEL
LIN {X 0,Y 157.489,Z 800.312,A -85,B 0,C 180,E1 21715.546,E2 21715.546} C_VEL
LIN {X 0,Y 169.885,Z 789.369,A -85,B 0,C 180,E1 21728.452,E2 21728.452} C_VEL
LIN {X 0,Y 187.609,Z 772.744,A -85,B 0,C 180,E1 21738.882,E2 21738.882} C_VEL
LIN {X 0,Y 201.349,Z 758.385,A -85,B 0,C 180,E1 21744.497,E2 21744.497} C_VEL
LIN {X 0,Y 201.875,Z 757.206,A -85,B 0,C 180,E1 21745.168,E2 21745.168} C_VEL
LIN {X 0,Y 176.431,Z 765.126,A -85,B 0,C 180,E1 21754.669,E2 21754.669} C_VEL
LIN {X 0,Y 157.796,Z 772.051,A -85,B 0,C 180,E1 21774.5,E2 21774.5} C_VEL
LIN {X 0,Y 159.696,Z 775.305,A -85,B 0,C 180,E1 21787.979,E2 21787.979} C_VEL
LIN {X 0,Y 166.812,Z 778.606,A -85,B 0,C 180,E1 21795.735,E2 21795.735} C_VEL
LIN {X 0,Y 173.075,Z 778.449,A -85,B 0,C 180,E1 21800.399,E2 21800.399} C_VEL
LIN {X 0,Y 183.61,Z 775.601,A -85,B 0,C 180,E1 21806.401,E2 21806.401} C_VEL
LIN {X 0,Y 200.716,Z 773.164,A -85,B 0,C 180,E1 21811.743,E2 21811.743} C_VEL
LIN {X 0,Y 199.478,Z 775.991,A -85,B 0,C 180,E1 21812.973,E2 21812.973} C_VEL
LIN {X 0,Y 179.452,Z 798.149,A -85,B 0,C 180,E1 21821.67,E2 21821.67} C_VEL
LIN {X 0,Y 163.151,Z 815.063,A -85,B 0,C 180,E1 21833.038,E2 21833.038} C_VEL
LIN {X 0,Y 153.238,Z 826.479,A -85,B 0,C 180,E1 21846.799,E2 21846.799} C_VEL
LIN {X 0,Y 150.521,Z 831.473,A -85,B 0,C 180,E1 21858.431,E2 21858.431} C_VEL
LIN {X 0,Y 150.869,Z 832.928,A -85,B 0,C 180,E1 21870.144,E2 21870.144} C_VEL
LIN {X 0,Y 150.574,Z 830.592,A -85,B 0,C 180,E1 21881.563,E2 21881.563} C_VEL
LIN {X 0,Y 153.961,Z 823.546,A -85,B 0,C 180,E1 21894.619,E2 21894.619} C_VEL
LIN {X 0,Y 164.416,Z 809.878,A -85,B 0,C 180,E1 21908.284,E2 21908.284} C_VEL
LIN {X 0,Y 181.078,Z 790.266,A -85,B 0,C 180,E1 21919.508,E2 21919.508} C_VEL
LIN {X 0,Y 187.691,Z 782.805,A -85,B 0,C 180,E1 21922.928,E2 21922.928} C_VEL
LIN {X 0,Y 172.915,Z 782.976,A -85,B 0,C 180,E1 21930.782,E2 21930.782} C_VEL
LIN {X 0,Y 161.283,Z 777.348,A -85,B 0,C 180,E1 21940.897,E2 21940.897} C_VEL
LIN {X 0,Y 155.492,Z 767.135,A -85,B 0,C 180,E1 21951.642,E2 21951.642} C_VEL
LIN {X 0,Y 169.634,Z 750.159,A -85,B 0,C 180,E1 21975.49,E2 21975.49} C_VEL
LIN {X 0,Y 193.409,Z 735.568,A -85,B 0,C 180,E1 21986.667,E2 21986.667} C_VEL
LIN {X 0,Y 219.035,Z 719.229,A -85,B 0,C 180,E1 21993.034,E2 21993.034} C_VEL
LIN {X 0,Y 222.094,Z 717.148,A -85,B 0,C 180,E1 21993.595,E2 21993.595} C_VEL
LIN {X 0,Y 222.203,Z 717.9,A -85,B 0,C 180,E1 21994.034,E2 21994.034} C_VEL
LIN {X 0,Y 203.345,Z 745.22,A -85,B 0,C 180,E1 21999.887,E2 21999.887} C_VEL
LIN {X 0,Y 189.619,Z 762.173,A -85,B 0,C 180,E1 22005.338,E2 22005.338} C_VEL
LIN {X 0,Y 178.706,Z 771.753,A -85,B 0,C 180,E1 22008.411,E2 22008.411} C_VEL
LIN {X 0,Y 167.995,Z 780.131,A -85,B 0,C 180,E1 22012.067,E2 22012.067} C_VEL
LIN {X 0,Y 153.911,Z 794.196,A -85,B 0,C 180,E1 22023.818,E2 22023.818} C_VEL
LIN {X 0,Y 145.617,Z 803.097,A -85,B 0,C 180,E1 22038.038,E2 22038.038} C_VEL
LIN {X 0,Y 143.589,Z 806.231,A -85,B 0,C 180,E1 22050.001,E2 22050.001} C_VEL
LIN {X 0,Y 144.027,Z 806.077,A -85,B 0,C 180,E1 22062.098,E2 22062.098} C_VEL
LIN {X 0,Y 148.51,Z 802.464,A -85,B 0,C 180,E1 22073.985,E2 22073.985} C_VEL
LIN {X 0,Y 158.895,Z 794,A -85,B 0,C 180,E1 22086.44,E2 22086.44} C_VEL
LIN {X 0,Y 174.96,Z 780.286,A -85,B 0,C 180,E1 22097.153,E2 22097.153} C_VEL
LIN {X 0,Y 191.726,Z 764.365,A -85,B 0,C 180,E1 22104.556,E2 22104.556} C_VEL
LIN {X 0,Y 191.882,Z 763.396,A -85,B 0,C 180,E1 22105.334,E2 22105.334} C_VEL
LIN {X 0,Y 165.707,Z 770.968,A -85,B 0,C 180,E1 22116.615,E2 22116.615} C_VEL
LIN {X 0,Y 151.261,Z 776.432,A -85,B 0,C 180,E1 22134.261,E2 22134.261} C_VEL
LIN {X 0,Y 154.592,Z 779.697,A -85,B 0,C 180,E1 22151.245,E2 22151.245} C_VEL
LIN {X 0,Y 173.924,Z 780.443,A -85,B 0,C 180,E1 22165.697,E2 22165.697} C_VEL
LIN {X 0,Y 191.172,Z 778.683,A -85,B 0,C 180,E1 22171.718,E2 22171.718} C_VEL
LIN {X 0,Y 187.87,Z 783.182,A -85,B 0,C 180,E1 22173.549,E2 22173.549} C_VEL
LIN {X 0,Y 168.016,Z 803.295,A -85,B 0,C 180,E1 22182.964,E2 22182.964} C_VEL
LIN {X 0,Y 151.988,Z 818.957,A -85,B 0,C 180,E1 22195.996,E2 22195.996} C_VEL
LIN {X 0,Y 143.904,Z 828.287,A -85,B 0,C 180,E1 22210.653,E2 22210.653} C_VEL
LIN {X 0,Y 142.349,Z 831.949,A -85,B 0,C 180,E1 22223.913,E2 22223.913} C_VEL
LIN {X 0,Y 143.018,Z 832.225,A -85,B 0,C 180,E1 22229.999,E2 22229.999} C_VEL
LIN {X 0,Y 142.728,Z 829.838,A -85,B 0,C 180,E1 22242.208,E2 22242.208} C_VEL
LIN {X 0,Y 146.557,Z 822.73,A -85,B 0,C 180,E1 22255.953,E2 22255.953} C_VEL
LIN {X 0,Y 158.108,Z 808.844,A -85,B 0,C 180,E1 22270.242,E2 22270.242} C_VEL
LIN {X 0,Y 175.679,Z 789.384,A -85,B 0,C 180,E1 22281.501,E2 22281.501} C_VEL
LIN {X 0,Y 178.188,Z 785.889,A -85,B 0,C 180,E1 22283.114,E2 22283.114} C_VEL
LIN {X 0,Y 162.154,Z 783.46,A -85,B 0,C 180,E1 22292.284,E2 22292.284} C_VEL
LIN {X 0,Y 149.621,Z 773.479,A -85,B 0,C 180,E1 22308.376,E2 22308.376} C_VEL
LIN {X 0,Y 161.983,Z 756.547,A -85,B 0,C 180,E1 22334.857,E2 22334.857} C_VEL
LIN {X 0,Y 183.085,Z 744.32,A -85,B 0,C 180,E1 22345.882,E2 22345.882} C_VEL
LIN {X 0,Y 209.104,Z 729.154,A -85,B 0,C 180,E1 22353.032,E2 22353.032} C_VEL
LIN {X 0,Y 212.079,Z 727.249,A -85,B 0,C 180,E1 22353.589,E2 22353.589} C_VEL
LIN {X 0,Y 193.817,Z 751.895,A -85,B 0,C 180,E1 22359.744,E2 22359.744} C_VEL
LIN {X 0,Y 173.893,Z 774.103,A -85,B 0,C 180,E1 22368.567,E2 22368.567} C_VEL
LIN {X 0,Y 167.995,Z 780.131,A -85,B 0,C 180,E1 22372.067,E2 22372.067} C_VEL
LIN {X 0,Y 157.663,Z 787.625,A -85,B 0,C 180,E1 22376.327,E2 22376.327} C_VEL
LIN {X 0,Y 147.978,Z 793.942,A -85,B 0,C 180,E1 22381.267,E2 22381.267} C_VEL
LIN {X 0,Y 139.125,Z 802.548,A -85,B 0,C 180,E1 22394.266,E2 22394.266} C_VEL
LIN {X 0,Y 136.427,Z 805.801,A -85,B 0,C 180,E1 22403.65,E2 22403.65} C_VEL
LIN {X 0,Y 135.465,Z 807.288,A -85,B 0,C 180,E1 22416.398,E2 22416.398} C_VEL
LIN {X 0,Y 139.356,Z 804.58,A -85,B 0,C 180,E1 22431.733,E2 22431.733} C_VEL
LIN {X 0,Y 150.938,Z 795.87,A -85,B 0,C 180,E1 22446.866,E2 22446.866} C_VEL
LIN {X 0,Y 167.447,Z 782.76,A -85,B 0,C 180,E1 22458.037,E2 22458.037} C_VEL
LIN {X 0,Y 181.219,Z 770.687,A -85,B 0,C 180,E1 22464.332,E2 22464.332} C_VEL
LIN {X 0,Y 182.472,Z 769.001,A -85,B 0,C 180,E1 22465.337,E2 22465.337} C_VEL
LIN {X 0,Y 164.499,Z 773.919,A -85,B 0,C 180,E1 22472.685,E2 22472.685} C_VEL
LIN {X 0,Y 144.573,Z 780.585,A -85,B 0,C 180,E1 22493.995,E2 22493.995} C_VEL
LIN {X 0,Y 148.056,Z 783.873,A -85,B 0,C 180,E1 22511.748,E2 22511.748} C_VEL
LIN {X 0,Y 167.962,Z 784.791,A -85,B 0,C 180,E1 22526.68,E2 22526.68} C_VEL
LIN {X 0,Y 181.701,Z 783.824,A -85,B 0,C 180,E1 22531.78,E2 22531.78} C_VEL
LIN {X 0,Y 161.285,Z 803.651,A -85,B 0,C 180,E1 22541.531,E2 22541.531} C_VEL
LIN {X 0,Y 144.579,Z 818.892,A -85,B 0,C 180,E1 22554.961,E2 22554.961} C_VEL
LIN {X 0,Y 135.995,Z 827.996,A -85,B 0,C 180,E1 22570.553,E2 22570.553} C_VEL
LIN {X 0,Y 134.474,Z 831.246,A -85,B 0,C 180,E1 22583.555,E2 22583.555} C_VEL
LIN {X 0,Y 135.12,Z 831.512,A -85,B 0,C 180,E1 22589.999,E2 22589.999} C_VEL
LIN {X 0,Y 134.894,Z 829.084,A -85,B 0,C 180,E1 22602.929,E2 22602.929} C_VEL
LIN {X 0,Y 140.004,Z 820.96,A -85,B 0,C 180,E1 22618.798,E2 22618.798} C_VEL
LIN {X 0,Y 151.49,Z 808.321,A -85,B 0,C 180,E1 22631.949,E2 22631.949} C_VEL
LIN {X 0,Y 168.826,Z 790.285,A -85,B 0,C 180,E1 22642.813,E2 22642.813} C_VEL
LIN {X 0,Y 167.407,Z 789.078,A -85,B 0,C 180,E1 22644.147,E2 22644.147} C_VEL
LIN {X 0,Y 147.45,Z 782.291,A -85,B 0,C 180,E1 22659.025,E2 22659.025} C_VEL
LIN {X 0,Y 147.411,Z 767.478,A -85,B 0,C 180,E1 22687.082,E2 22687.082} C_VEL
LIN {X 0,Y 169.588,Z 753.992,A -85,B 0,C 180,E1 22703.617,E2 22703.617} C_VEL
LIN {X 0,Y 194.053,Z 741.088,A -85,B 0,C 180,E1 22711.806,E2 22711.806} C_VEL
LIN {X 0,Y 201.342,Z 737.106,A -85,B 0,C 180,E1 22713.58,E2 22713.58} C_VEL
LIN {X 0,Y 182.758,Z 759.789,A -85,B 0,C 180,E1 22720.197,E2 22720.197} C_VEL
LIN {X 0,Y 163.054,Z 779.897,A -85,B 0,C 180,E1 22729.618,E2 22729.618} C_VEL
LIN {X 0,Y 147.978,Z 793.942,A -85,B 0,C 180,E1 22741.267,E2 22741.267} C_VEL
LIN {X 0,Y 139.239,Z 799.261,A -85,B 0,C 180,E1 22746.947,E2 22746.947} C_VEL
LIN {X 0,Y 131.513,Z 803.341,A -85,B 0,C 180,E1 22753.411,E2 22753.411} C_VEL
LIN {X 0,Y 128.616,Z 806.532,A -85,B 0,C 180,E1 22763.263,E2 22763.263} C_VEL
LIN {X 0,Y 127.621,Z 807.993,A -85,B 0,C 180,E1 22776.793,E2 22776.793} C_VEL
LIN {X 0,Y 130.701,Z 806.099,A -85,B 0,C 180,E1 22790.269,E2 22790.269} C_VEL
LIN {X 0,Y 141.189,Z 798.966,A -85,B 0,C 180,E1 22805.636,E2 22805.636} C_VEL
LIN {X 0,Y 158.372,Z 786.41,A -85,B 0,C 180,E1 22818.148,E2 22818.148} C_VEL
LIN {X 0,Y 171.123,Z 776.173,A -85,B 0,C 180,E1 22824.237,E2 22824.237} C_VEL
LIN {X 0,Y 172.636,Z 774.362,A -85,B 0,C 180,E1 22825.468,E2 22825.468} C_VEL
LIN {X 0,Y 150.864,Z 779.878,A -85,B 0,C 180,E1 22836.401,E2 22836.401} C_VEL
LIN {X 0,Y 137.153,Z 785.757,A -85,B 0,C 180,E1 22859.986,E2 22859.986} C_VEL
LIN {X 0,Y 146.514,Z 788.531,A -85,B 0,C 180,E1 22877.984,E2 22877.984} C_VEL
LIN {X 0,Y 161.946,Z 788.942,A -85,B 0,C 180,E1 22887.755,E2 22887.755} C_VEL
LIN {X 0,Y 172.062,Z 788.482,A -85,B 0,C 180,E1 22891.737,E2 22891.737} C_VEL
LIN {X 0,Y 151.733,Z 806.507,A -85,B 0,C 180,E1 22901.756,E2 22901.756} C_VEL
LIN {X 0,Y 135.286,Z 820.444,A -85,B 0,C 180,E1 22916.097,E2 22916.097} C_VEL
LIN {X 0,Y 128.116,Z 827.677,A -85,B 0,C 180,E1 22930.393,E2 22930.393} C_VEL
LIN {X 0,Y 126.569,Z 830.54,A -85,B 0,C 180,E1 22943.151,E2 22943.151} C_VEL
LIN {X 0,Y 127.236,Z 830.801,A -85,B 0,C 180,E1 22949.999,E2 22949.999} C_VEL
LIN {X 0,Y 127.081,Z 828.331,A -85,B 0,C 180,E1 22963.739,E2 22963.739} C_VEL
LIN {X 0,Y 132.758,Z 820.262,A -85,B 0,C 180,E1 22980.299,E2 22980.299} C_VEL
LIN {X 0,Y 146.462,Z 806.449,A -85,B 0,C 180,E1 22994.908,E2 22994.908} C_VEL
LIN {X 0,Y 159.631,Z 793.624,A -85,B 0,C 180,E1 23003.005,E2 23003.005} C_VEL
LIN {X 0,Y 159.433,Z 792.617,A -85,B 0,C 180,E1 23003.916,E2 23003.916} C_VEL
LIN {X 0,Y 139.146,Z 785.193,A -85,B 0,C 180,E1 23021.028,E2 23021.028} C_VEL
LIN {X 0,Y 144.734,Z 769.377,A -85,B 0,C 180,E1 23052.05,E2 23052.05} C_VEL
LIN {X 0,Y 171.345,Z 755.436,A -85,B 0,C 180,E1 23067.73,E2 23067.73} C_VEL
LIN {X 0,Y 191.228,Z 745.564,A -85,B 0,C 180,E1 23073.543,E2 23073.543} C_VEL
LIN {X 0,Y 170.422,Z 768.197,A -85,B 0,C 180,E1 23081.175,E2 23081.175} C_VEL
LIN {X 0,Y 151.309,Z 785.977,A -85,B 0,C 180,E1 23091.438,E2 23091.438} C_VEL
LIN {X 0,Y 137.332,Z 798.038,A -85,B 0,C 180,E1 23103.925,E2 23103.925} C_VEL
LIN {X 0,Y 131.513,Z 803.341,A -85,B 0,C 180,E1 23113.411,E2 23113.411} C_VEL
LIN {X 0,Y 126.948,Z 805.685,A -85,B 0,C 180,E1 23118.798,E2 23118.798} C_VEL
LIN {X 0,Y 120.138,Z 808.077,A -85,B 0,C 180,E1 23127.427,E2 23127.427} C_VEL
LIN {X 0,Y 119.992,Z 808.155,A -85,B 0,C 180,E1 23128.476,E2 23128.476} C_VEL
LIN {X 0,Y 120.847,Z 808.181,A -85,B 0,C 180,E1 23144.465,E2 23144.465} C_VEL
LIN {X 0,Y 129.294,Z 803.051,A -85,B 0,C 180,E1 23161.687,E2 23161.687} C_VEL
LIN {X 0,Y 146.062,Z 792.085,A -85,B 0,C 180,E1 23176.327,E2 23176.327} C_VEL
LIN {X 0,Y 163.067,Z 779.31,A -85,B 0,C 180,E1 23185.482,E2 23185.482} C_VEL
LIN {X 0,Y 138.29,Z 785.339,A -85,B 0,C 180,E1 23200.876,E2 23200.876} C_VEL
LIN {X 0,Y 131.352,Z 790.705,A -85,B 0,C 180,E1 23226.582,E2 23226.582} C_VEL
LIN {X 0,Y 147.11,Z 792.745,A -85,B 0,C 180,E1 23244.21,E2 23244.21} C_VEL
LIN {X 0,Y 161.72,Z 792.713,A -85,B 0,C 180,E1 23251.35,E2 23251.35} C_VEL
LIN {X 0,Y 142.137,Z 809.075,A -85,B 0,C 180,E1 23261.99,E2 23261.99} C_VEL
LIN {X 0,Y 126.828,Z 821.188,A -85,B 0,C 180,E1 23276.367,E2 23276.367} C_VEL
LIN {X 0,Y 119.645,Z 827.963,A -85,B 0,C 180,E1 23292.519,E2 23292.519} C_VEL
LIN {X 0,Y 118.681,Z 829.834,A -85,B 0,C 180,E1 23302.693,E2 23302.693} C_VEL
LIN {X 0,Y 119.34,Z 830.087,A -85,B 0,C 180,E1 23309.999,E2 23309.999} C_VEL
LIN {X 0,Y 119.298,Z 827.575,A -85,B 0,C 180,E1 23324.654,E2 23324.654} C_VEL
LIN {X 0,Y 125.242,Z 819.97,A -85,B 0,C 180,E1 23341.353,E2 23341.353} C_VEL
LIN {X 0,Y 139.806,Z 806.348,A -85,B 0,C 180,E1 23356.613,E2 23356.613} C_VEL
LIN {X 0,Y 150.58,Z 796.598,A -85,B 0,C 180,E1 23363.3,E2 23363.3} C_VEL
LIN {X 0,Y 140.335,Z 792.925,A -85,B 0,C 180,E1 23371.076,E2 23371.076} C_VEL
LIN {X 0,Y 129.248,Z 782.322,A -85,B 0,C 180,E1 23396.153,E2 23396.153} C_VEL
LIN {X 0,Y 150.713,Z 767.39,A -85,B 0,C 180,E1 23422.068,E2 23422.068} C_VEL
LIN {X 0,Y 180.328,Z 753.856,A -85,B 0,C 180,E1 23433.426,E2 23433.426} C_VEL
LIN {X 0,Y 160.474,Z 773.627,A -85,B 0,C 180,E1 23441.206,E2 23441.206} C_VEL
LIN {X 0,Y 141.405,Z 789.979,A -85,B 0,C 180,E1 23452.145,E2 23452.145} C_VEL
LIN {X 0,Y 127.837,Z 800.792,A -85,B 0,C 180,E1 23465.596,E2 23465.596} C_VEL
LIN {X 0,Y 120.804,Z 807.266,A -85,B 0,C 180,E1 23482.825,E2 23482.825} C_VEL
LIN {X 0,Y 119.992,Z 808.155,A -85,B 0,C 180,E1 23488.476,E2 23488.476} C_VEL
LIN {X 0,Y 117.389,Z 809.052,A -85,B 0,C 180,E1 23494.654,E2 23494.654} C_VEL
LIN {X 0,Y 113.034,Z 809.06,A -85,B 0,C 180,E1 23504.364,E2 23504.364} C_VEL
LIN {X 0,Y 113.177,Z 808.88,A -85,B 0,C 180,E1 23505.482,E2 23505.482} C_VEL
LIN {X 0,Y 122.54,Z 803.743,A -85,B 0,C 180,E1 23523.658,E2 23523.658} C_VEL
LIN {X 0,Y 140.65,Z 792.774,A -85,B 0,C 180,E1 23538.688,E2 23538.688} C_VEL
LIN {X 0,Y 151.781,Z 785.274,A -85,B 0,C 180,E1 23544.484,E2 23544.484} C_VEL
LIN {X 0,Y 152.58,Z 784.108,A -85,B 0,C 180,E1 23545.902,E2 23545.902} C_VEL
LIN {X 0,Y 126.682,Z 790.504,A -85,B 0,C 180,E1 23566.201,E2 23566.201} C_VEL
LIN {X 0,Y 127.777,Z 795.206,A -85,B 0,C 180,E1 23593.646,E2 23593.646} C_VEL
LIN {X 0,Y 151.54,Z 796.615,A -85,B 0,C 180,E1 23611.032,E2 23611.032} C_VEL
LIN {X 0,Y 151.341,Z 797.396,A -85,B 0,C 180,E1 23611.797,E2 23611.797} C_VEL
LIN {X 0,Y 130.246,Z 813.068,A -85,B 0,C 180,E1 23624.019,E2 23624.019} C_VEL
LIN {X 0,Y 116.894,Z 822.897,A -85,B 0,C 180,E1 23638.906,E2 23638.906} C_VEL
LIN {X 0,Y 111.443,Z 827.921,A -85,B 0,C 180,E1 23654.284,E2 23654.284} C_VEL
LIN {X 0,Y 111.45,Z 829.375,A -85,B 0,C 180,E1 23669.999,E2 23669.999} C_VEL
LIN {X 0,Y 111.54,Z 826.821,A -85,B 0,C 180,E1 23685.699,E2 23685.699} C_VEL
LIN {X 0,Y 118.332,Z 819.14,A -85,B 0,C 180,E1 23703.414,E2 23703.414} C_VEL
LIN {X 0,Y 134.643,Z 805.146,A -85,B 0,C 180,E1 23719.413,E2 23719.413} C_VEL
LIN {X 0,Y 140.295,Z 800.383,A -85,B 0,C 180,E1 23722.948,E2 23722.948} C_VEL
LIN {X 0,Y 141.125,Z 798.574,A -85,B 0,C 180,E1 23724.614,E2 23724.614} C_VEL
LIN {X 0,Y 122.28,Z 789.015,A -85,B 0,C 180,E1 23749.352,E2 23749.352} C_VEL
LIN {X 0,Y 138.215,Z 774.817,A -85,B 0,C 180,E1 23779.135,E2 23779.135} C_VEL
LIN {X 0,Y 169.094,Z 761.579,A -85,B 0,C 180,E1 23793.165,E2 23793.165} C_VEL
LIN {X 0,Y 167.074,Z 764.037,A -85,B 0,C 180,E1 23794.55,E2 23794.55} C_VEL
LIN {X 0,Y 145.849,Z 782.563,A -85,B 0,C 180,E1 23803.589,E2 23803.589} C_VEL
LIN {X 0,Y 127.976,Z 796.219,A -85,B 0,C 180,E1 23815.935,E2 23815.935} C_VEL
LIN {X 0,Y 116.541,Z 804.832,A -85,B 0,C 180,E1 23831.112,E2 23831.112} C_VEL
LIN {X 0,Y 112.128,Z 808.878,A -85,B 0,C 180,E1 23848.371,E2 23848.371} C_VEL
LIN {X 0,Y 113.177,Z 808.88,A -85,B 0,C 180,E1 23865.482,E2 23865.482} C_VEL
LIN {X 0,Y 112.438,Z 807.688,A -85,B 0,C 180,E1 23874.371,E2 23874.371} C_VEL
LIN {X 0,Y 113.834,Z 805.531,A -85,B 0,C 180,E1 23883.215,E2 23883.215} C_VEL
LIN {X 0,Y 130.954,Z 796.164,A -85,B 0,C 180,E1 23898.513,E2 23898.513} C_VEL
LIN {X 0,Y 143.399,Z 788.265,A -85,B 0,C 180,E1 23905.835,E2 23905.835} C_VEL
LIN {X 0,Y 116.774,Z 795.188,A -85,B 0,C 180,E1 23932.558,E2 23932.558} C_VEL
LIN {X 0,Y 120.848,Z 798.547,A -85,B 0,C 180,E1 23954.445,E2 23954.445} C_VEL
LIN {X 0,Y 137.245,Z 799.957,A -85,B 0,C 180,E1 23968.391,E2 23968.391} C_VEL
LIN {X 0,Y 141.559,Z 800.723,A -85,B 0,C 180,E1 23971.47,E2 23971.47} C_VEL
LIN {X 0,Y 119.149,Z 816.024,A -85,B 0,C 180,E1 23985.839,E2 23985.839} C_VEL
LIN {X 0,Y 105.971,Z 825.169,A -85,B 0,C 180,E1 24004.706,E2 24004.706} C_VEL
LIN {X 0,Y 102.877,Z 828.41,A -85,B 0,C 180,E1 24021.563,E2 24021.563} C_VEL
LIN {X 0,Y 103.541,Z 828.661,A -85,B 0,C 180,E1 24029.998,E2 24029.998} C_VEL
LIN {X 0,Y 103.807,Z 826.063,A -85,B 0,C 180,E1 24046.902,E2 24046.902} C_VEL
LIN {X 0,Y 111.641,Z 818.255,A -85,B 0,C 180,E1 24065.836,E2 24065.836} C_VEL
LIN {X 0,Y 129.189,Z 804.411,A -85,B 0,C 180,E1 24082.047,E2 24082.047} C_VEL
LIN {X 0,Y 132.657,Z 801.312,A -85,B 0,C 180,E1 24084.605,E2 24084.605} C_VEL
LIN {X 0,Y 115.039,Z 791.432,A -85,B 0,C 180,E1 24112.48,E2 24112.48} C_VEL
LIN {X 0,Y 135.784,Z 777.323,A -85,B 0,C 180,E1 24142.906,E2 24142.906} C_VEL
LIN {X 0,Y 158.313,Z 768.446,A -85,B 0,C 180,E1 24152.979,E2 24152.979} C_VEL
LIN {X 0,Y 158.139,Z 769.15,A -85,B 0,C 180,E1 24153.845,E2 24153.845} C_VEL
LIN {X 0,Y 135.821,Z 786.962,A -85,B 0,C 180,E1 24163.761,E2 24163.761} C_VEL
LIN {X 0,Y 116.558,Z 800.436,A -85,B 0,C 180,E1 24178.809,E2 24178.809} C_VEL
LIN {X 0,Y 107.409,Z 806.874,A -85,B 0,C 180,E1 24193.681,E2 24193.681} C_VEL
LIN {X 0,Y 104.246,Z 809.833,A -85,B 0,C 180,E1 24210.002,E2 24210.002} C_VEL
LIN {X 0,Y 105.529,Z 809.586,A -85,B 0,C 180,E1 24226.622,E2 24226.622} C_VEL
LIN {X 0,Y 113.834,Z 805.531,A -85,B 0,C 180,E1 24243.215,E2 24243.215} C_VEL
LIN {X 0,Y 117.304,Z 802.484,A -85,B 0,C 180,E1 24251.611,E2 24251.611} C_VEL
LIN {X 0,Y 122.768,Z 798.476,A -85,B 0,C 180,E1 24259.35,E2 24259.35} C_VEL
LIN {X 0,Y 133.965,Z 792.209,A -85,B 0,C 180,E1 24265.703,E2 24265.703} C_VEL
LIN {X 0,Y 109.59,Z 798.275,A -85,B 0,C 180,E1 24292.067,E2 24292.067} C_VEL
LIN {X 0,Y 113.859,Z 801.684,A -85,B 0,C 180,E1 24315.353,E2 24315.353} C_VEL
LIN {X 0,Y 131.945,Z 803.35,A -85,B 0,C 180,E1 24330.626,E2 24330.626} C_VEL
LIN {X 0,Y 111.234,Z 816.571,A -85,B 0,C 180,E1 24344.852,E2 24344.852} C_VEL
LIN {X 0,Y 98.688,Z 824.461,A -85,B 0,C 180,E1 24362.69,E2 24362.69} C_VEL
LIN {X 0,Y 94.984,Z 827.696,A -85,B 0,C 180,E1 24380.856,E2 24380.856} C_VEL
LIN {X 0,Y 95.641,Z 827.948,A -85,B 0,C 180,E1 24389.998,E2 24389.998} C_VEL
LIN {X 0,Y 96.566,Z 824.764,A -85,B 0,C 180,E1 24410.404,E2 24410.404} C_VEL
LIN {X 0,Y 107.187,Z 815.901,A -85,B 0,C 180,E1 24431.062,E2 24431.062} C_VEL
LIN {X 0,Y 121.899,Z 805.259,A -85,B 0,C 180,E1 24443.583,E2 24443.583} C_VEL
LIN {X 0,Y 123.199,Z 803.62,A -85,B 0,C 180,E1 24445.309,E2 24445.309} C_VEL
LIN {X 0,Y 108.121,Z 793.633,A -85,B 0,C 180,E1 24476.017,E2 24476.017} C_VEL
LIN {X 0,Y 133.943,Z 779.633,A -85,B 0,C 180,E1 24506.802,E2 24506.802} C_VEL
LIN {X 0,Y 148.009,Z 774.573,A -85,B 0,C 180,E1 24512.923,E2 24512.923} C_VEL
LIN {X 0,Y 137.024,Z 783.187,A -85,B 0,C 180,E1 24518.011,E2 24518.011} C_VEL
LIN {X 0,Y 117.209,Z 796.604,A -85,B 0,C 180,E1 24529.926,E2 24529.926} C_VEL
LIN {X 0,Y 101.775,Z 806.352,A -85,B 0,C 180,E1 24548.242,E2 24548.242} C_VEL
LIN {X 0,Y 97.441,Z 809.459,A -85,B 0,C 180,E1 24561.092,E2 24561.092} C_VEL
LIN {X 0,Y 96.375,Z 810.553,A -85,B 0,C 180,E1 24570.002,E2 24570.002} C_VEL
LIN {X 0,Y 97.941,Z 810.29,A -85,B 0,C 180,E1 24587.951,E2 24587.951} C_VEL
LIN {X 0,Y 109.553,Z 805.13,A -85,B 0,C 180,E1 24608.311,E2 24608.311} C_VEL
LIN {X 0,Y 122.768,Z 798.476,A -85,B 0,C 180,E1 24619.35,E2 24619.35} C_VEL
LIN {X 0,Y 124.207,Z 796.941,A -85,B 0,C 180,E1 24622.582,E2 24622.582} C_VEL
LIN {X 0,Y 120.314,Z 796.593,A -85,B 0,C 180,E1 24628.268,E2 24628.268} C_VEL
LIN {X 0,Y 117.866,Z 796.973,A -85,B 0,C 180,E1 24630.344,E2 24630.344} C_VEL
LIN {X 0,Y 101.418,Z 802.388,A -85,B 0,C 180,E1 24659.98,E2 24659.98} C_VEL
LIN {X 0,Y 113.171,Z 805.46,A -85,B 0,C 180,E1 24683.56,E2 24683.56} C_VEL
LIN {X 0,Y 122.555,Z 806.167,A -85,B 0,C 180,E1 24690.456,E2 24690.456} C_VEL
LIN {X 0,Y 100.029,Z 818.925,A -85,B 0,C 180,E1 24707.244,E2 24707.244} C_VEL
LIN {X 0,Y 88.413,Z 825.79,A -85,B 0,C 180,E1 24730.036,E2 24730.036} C_VEL
LIN {X 0,Y 87.727,Z 827.233,A -85,B 0,C 180,E1 24749.998,E2 24749.998} C_VEL
LIN {X 0,Y 88.508,Z 824.546,A -85,B 0,C 180,E1 24769.938,E2 24769.938} C_VEL
LIN {X 0,Y 99.591,Z 816.058,A -85,B 0,C 180,E1 24792.401,E2 24792.401} C_VEL
LIN {X 0,Y 112.296,Z 807.608,A -85,B 0,C 180,E1 24803.739,E2 24803.739} C_VEL
LIN {X 0,Y 113.68,Z 805.78,A -85,B 0,C 180,E1 24806.119,E2 24806.119} C_VEL
LIN {X 0,Y 101.681,Z 795.664,A -85,B 0,C 180,E1 24840.019,E2 24840.019} C_VEL
LIN {X 0,Y 131.208,Z 782.372,A -85,B 0,C 180,E1 24870.073,E2 24870.073} C_VEL
LIN {X 0,Y 137.34,Z 780.345,A -85,B 0,C 180,E1 24872.736,E2 24872.736} C_VEL
LIN {X 0,Y 120.487,Z 791.846,A -85,B 0,C 180,E1 24881.278,E2 24881.278} C_VEL
LIN {X 0,Y 99.972,Z 803.927,A -85,B 0,C 180,E1 24898.107,E2 24898.107} C_VEL
LIN {X 0,Y 89.683,Z 810.191,A -85,B 0,C 180,E1 24920.314,E2 24920.314} C_VEL
LIN {X 0,Y 88.493,Z 811.274,A -85,B 0,C 180,E1 24930.002,E2 24930.002} C_VEL
LIN {X 0,Y 90.422,Z 810.993,A -85,B 0,C 180,E1 24949.502,E2 24949.502} C_VEL
LIN {X 0,Y 103.383,Z 805.822,A -85,B 0,C 180,E1 24971.066,E2 24971.066} C_VEL
LIN {X 0,Y 120.918,Z 797.544,A -85,B 0,C 180,E1 24984.222,E2 24984.222} C_VEL
LIN {X 0,Y 123.318,Z 795.957,A -85,B 0,C 180,E1 24986.569,E2 24986.569} C_VEL
LIN {X 0,Y 117.866,Z 796.973,A -85,B 0,C 180,E1 24990.344,E2 24990.344} C_VEL
LIN {X 0,Y 106.454,Z 800.097,A -85,B 0,C 180,E1 24996.938,E2 24996.938} C_VEL
LIN {X 0,Y 97.789,Z 802.732,A -85,B 0,C 180,E1 25003.838,E2 25003.838} C_VEL
LIN {X 0,Y 97.111,Z 802.951,A -85,B 0,C 180,E1 25005.045,E2 25005.045} C_VEL
LIN {X 0,Y 99.709,Z 807.338,A -85,B 0,C 180,E1 25037.598,E2 25037.598} C_VEL
LIN {X 0,Y 111.987,Z 808.641,A -85,B 0,C 180,E1 25049.505,E2 25049.505} C_VEL
LIN {X 0,Y 105.462,Z 812.498,A -85,B 0,C 180,E1 25054.354,E2 25054.354} C_VEL
LIN {X 0,Y 87.165,Z 821.682,A -85,B 0,C 180,E1 25072.874,E2 25072.874} C_VEL
LIN {X 0,Y 80.627,Z 825.265,A -85,B 0,C 180,E1 25089.29,E2 25089.29} C_VEL
LIN {X 0,Y 79.817,Z 826.519,A -85,B 0,C 180,E1 25109.998,E2 25109.998} C_VEL
LIN {X 0,Y 80.966,Z 823.784,A -85,B 0,C 180,E1 25131.886,E2 25131.886} C_VEL
LIN {X 0,Y 94.068,Z 814.997,A -85,B 0,C 180,E1 25156.214,E2 25156.214} C_VEL
LIN {X 0,Y 104.993,Z 807.968,A -85,B 0,C 180,E1 25166.293,E2 25166.293} C_VEL
LIN {X 0,Y 95.804,Z 797.589,A -85,B 0,C 180,E1 25204.538,E2 25204.538} C_VEL
LIN {X 0,Y 123.025,Z 786.793,A -85,B 0,C 180,E1 25230.831,E2 25230.831} C_VEL
LIN {X 0,Y 126.184,Z 786.121,A -85,B 0,C 180,E1 25233.156,E2 25233.156} C_VEL
LIN {X 0,Y 101.695,Z 800.43,A -85,B 0,C 180,E1 25247.437,E2 25247.437} C_VEL
LIN {X 0,Y 84.984,Z 809.137,A -85,B 0,C 180,E1 25269.198,E2 25269.198} C_VEL
LIN {X 0,Y 80.618,Z 811.994,A -85,B 0,C 180,E1 25290.002,E2 25290.002} C_VEL
LIN {X 0,Y 82.97,Z 811.696,A -85,B 0,C 180,E1 25311.335,E2 25311.335} C_VEL
LIN {X 0,Y 97.47,Z 806.509,A -85,B 0,C 180,E1 25334.17,E2 25334.17} C_VEL
LIN {X 0,Y 112.738,Z 799.942,A -85,B 0,C 180,E1 25345.426,E2 25345.426} C_VEL
LIN {X 0,Y 113.7,Z 799.279,A -85,B 0,C 180,E1 25346.843,E2 25346.843} C_VEL
LIN {X 0,Y 97.111,Z 802.951,A -85,B 0,C 180,E1 25365.045,E2 25365.045} C_VEL
LIN {X 0,Y 90.515,Z 805.649,A -85,B 0,C 180,E1 25374.81,E2 25374.81} C_VEL
LIN {X 0,Y 87.118,Z 808.226,A -85,B 0,C 180,E1 25385.724,E2 25385.724} C_VEL
LIN {X 0,Y 101.6,Z 810.886,A -85,B 0,C 180,E1 25408.606,E2 25408.606} C_VEL
LIN {X 0,Y 99.207,Z 812.679,A -85,B 0,C 180,E1 25411.648,E2 25411.648} C_VEL
LIN {X 0,Y 77.781,Z 822.323,A -85,B 0,C 180,E1 25434.4,E2 25434.4} C_VEL
LIN {X 0,Y 71.417,Z 825.551,A -85,B 0,C 180,E1 25457.798,E2 25457.798} C_VEL
LIN {X 0,Y 71.904,Z 825.804,A -85,B 0,C 180,E1 25469.998,E2 25469.998} C_VEL
LIN {X 0,Y 73.517,Z 823.021,A -85,B 0,C 180,E1 25494.238,E2 25494.238} C_VEL
LIN {X 0,Y 86.47,Z 815.303,A -85,B 0,C 180,E1 25517.879,E2 25517.879} C_VEL
LIN {X 0,Y 94.795,Z 810.752,A -85,B 0,C 180,E1 25525.4,E2 25525.4} C_VEL
LIN {X 0,Y 95.669,Z 809.743,A -85,B 0,C 180,E1 25527.163,E2 25527.163} C_VEL
LIN {X 0,Y 90.543,Z 799.354,A -85,B 0,C 180,E1 25569.616,E2 25569.616} C_VEL
LIN {X 0,Y 114.838,Z 790.866,A -85,B 0,C 180,E1 25591.73,E2 25591.73} C_VEL
LIN {X 0,Y 115.241,Z 791.036,A -85,B 0,C 180,E1 25592.905,E2 25592.905} C_VEL
LIN {X 0,Y 91.047,Z 803.633,A -85,B 0,C 180,E1 25608.471,E2 25608.471} C_VEL
LIN {X 0,Y 77.681,Z 809.889,A -85,B 0,C 180,E1 25627.137,E2 25627.137} C_VEL
LIN {X 0,Y 72.731,Z 812.715,A -85,B 0,C 180,E1 25650.002,E2 25650.002} C_VEL
LIN {X 0,Y 75.633,Z 812.399,A -85,B 0,C 180,E1 25673.523,E2 25673.523} C_VEL
LIN {X 0,Y 91.616,Z 807.293,A -85,B 0,C 180,E1 25697.405,E2 25697.405} C_VEL
LIN {X 0,Y 101.477,Z 803.537,A -85,B 0,C 180,E1 25704.884,E2 25704.884} C_VEL
LIN {X 0,Y 103.583,Z 802.444,A -85,B 0,C 180,E1 25707.528,E2 25707.528} C_VEL
LIN {X 0,Y 87.118,Z 808.226,A -85,B 0,C 180,E1 25745.724,E2 25745.724} C_VEL
LIN {X 0,Y 87.302,Z 810.683,A -85,B 0,C 180,E1 25757.176,E2 25757.176} C_VEL
LIN {X 0,Y 90.648,Z 813.193,A -85,B 0,C 180,E1 25768.223,E2 25768.223} C_VEL
LIN {X 0,Y 91.773,Z 813.407,A -85,B 0,C 180,E1 25769.532,E2 25769.532} C_VEL
LIN {X 0,Y 71.319,Z 821.608,A -85,B 0,C 180,E1 25790.59,E2 25790.59} C_VEL
LIN {X 0,Y 63.602,Z 824.834,A -85,B 0,C 180,E1 25816.271,E2 25816.271} C_VEL
LIN {X 0,Y 63.983,Z 825.089,A -85,B 0,C 180,E1 25829.998,E2 25829.998} C_VEL
LIN {X 0,Y 66.24,Z 822.261,A -85,B 0,C 180,E1 25857.105,E2 25857.105} C_VEL
LIN {X 0,Y 82.916,Z 813.623,A -85,B 0,C 180,E1 25883.813,E2 25883.813} C_VEL
LIN {X 0,Y 86.286,Z 811.272,A -85,B 0,C 180,E1 25888.382,E2 25888.382} C_VEL
LIN {X 0,Y 89.561,Z 799.641,A -85,B 0,C 180,E1 25939.717,E2 25939.717} C_VEL
LIN {X 0,Y 104.448,Z 795.216,A -85,B 0,C 180,E1 25951.593,E2 25951.593} C_VEL
LIN {X 0,Y 100.681,Z 797.279,A -85,B 0,C 180,E1 25954.472,E2 25954.472} C_VEL
LIN {X 0,Y 76.91,Z 807.941,A -85,B 0,C 180,E1 25973.939,E2 25973.939} C_VEL
LIN {X 0,Y 66.537,Z 812.389,A -85,B 0,C 180,E1 25996.893,E2 25996.893} C_VEL
LIN {X 0,Y 64.853,Z 813.434,A -85,B 0,C 180,E1 26010.002,E2 26010.002} C_VEL
LIN {X 0,Y 70.324,Z 812.617,A -85,B 0,C 180,E1 26040.815,E2 26040.815} C_VEL
LIN {X 0,Y 85.929,Z 808.138,A -85,B 0,C 180,E1 26060.914,E2 26060.914} C_VEL
LIN {X 0,Y 93.141,Z 805.68,A -85,B 0,C 180,E1 26066.297,E2 26066.297} C_VEL
LIN {X 0,Y 94.087,Z 805.256,A -85,B 0,C 180,E1 26067.752,E2 26067.752} C_VEL
LIN {X 0,Y 80.654,Z 810.952,A -85,B 0,C 180,E1 26110.759,E2 26110.759} C_VEL
LIN {X 0,Y 90.648,Z 813.193,A -85,B 0,C 180,E1 26128.223,E2 26128.223} C_VEL
LIN {X 0,Y 89.952,Z 814.401,A -85,B 0,C 180,E1 26131.373,E2 26131.373} C_VEL
LIN {X 0,Y 82.424,Z 816.967,A -85,B 0,C 180,E1 26135.733,E2 26135.733} C_VEL
LIN {X 0,Y 66.881,Z 820.388,A -85,B 0,C 180,E1 26143.86,E2 26143.86} C_VEL
LIN {X 0,Y 65.381,Z 820.827,A -85,B 0,C 180,E1 26145.758,E2 26145.758} C_VEL
LIN {X 0,Y 55.846,Z 824.117,A -85,B 0,C 180,E1 26174.319,E2 26174.319} C_VEL
LIN {X 0,Y 56.031,Z 824.371,A -85,B 0,C 180,E1 26189.997,E2 26189.997} C_VEL
LIN {X 0,Y 59.13,Z 821.494,A -85,B 0,C 180,E1 26220.692,E2 26220.692} C_VEL
LIN {X 0,Y 76.066,Z 813.799,A -85,B 0,C 180,E1 26246.734,E2 26246.734} C_VEL
LIN {X 0,Y 77.15,Z 812.72,A -85,B 0,C 180,E1 26249.581,E2 26249.581} C_VEL
LIN {X 0,Y 82.458,Z 802.402,A -85,B 0,C 180,E1 26301.496,E2 26301.496} C_VEL
LIN {X 0,Y 93.15,Z 799.418,A -85,B 0,C 180,E1 26310.859,E2 26310.859} C_VEL
LIN {X 0,Y 87.863,Z 801.939,A -85,B 0,C 180,E1 26315.328,E2 26315.328} C_VEL
LIN {X 0,Y 66.782,Z 810.153,A -85,B 0,C 180,E1 26335.603,E2 26335.603} C_VEL
LIN {X 0,Y 58.902,Z 813.118,A -85,B 0,C 180,E1 26355.157,E2 26355.157} C_VEL
LIN {X 0,Y 56.97,Z 814.152,A -85,B 0,C 180,E1 26370.003,E2 26370.003} C_VEL
LIN {X 0,Y 61.358,Z 813.805,A -85,B 0,C 180,E1 26399.47,E2 26399.47} C_VEL
LIN {X 0,Y 80.221,Z 809.097,A -85,B 0,C 180,E1 26424.602,E2 26424.602} C_VEL
LIN {X 0,Y 83.73,Z 808.06,A -85,B 0,C 180,E1 26427.242,E2 26427.242} C_VEL
LIN {X 0,Y 81.517,Z 814.758,A -85,B 0,C 180,E1 26487.54,E2 26487.54} C_VEL
LIN {X 0,Y 79.108,Z 816.073,A -85,B 0,C 180,E1 26490.849,E2 26490.849} C_VEL
LIN {X 0,Y 65.381,Z 820.827,A -85,B 0,C 180,E1 26505.758,E2 26505.758} C_VEL
LIN {X 0,Y 57.659,Z 822.507,A -85,B 0,C 180,E1 26515.511,E2 26515.511} C_VEL
LIN {X 0,Y 47.634,Z 823.474,A -85,B 0,C 180,E1 26537.121,E2 26537.121} C_VEL
LIN {X 0,Y 48.098,Z 823.654,A -85,B 0,C 180,E1 26549.997,E2 26549.997} C_VEL
LIN {X 0,Y 52.321,Z 820.729,A -85,B 0,C 180,E1 26585.228,E2 26585.228} C_VEL
LIN {X 0,Y 66.199,Z 815.224,A -85,B 0,C 180,E1 26607.262,E2 26607.262} C_VEL
LIN {X 0,Y 68.061,Z 814.033,A -85,B 0,C 180,E1 26611.022,E2 26611.022} C_VEL
LIN {X 0,Y 82.637,Z 803.017,A -85,B 0,C 180,E1 26670.501,E2 26670.501} C_VEL
LIN {X 0,Y 77.769,Z 804.954,A -85,B 0,C 180,E1 26674.441,E2 26674.441} C_VEL
LIN {X 0,Y 56.644,Z 812.144,A -85,B 0,C 180,E1 26697.804,E2 26697.804} C_VEL
LIN {X 0,Y 49.088,Z 814.868,A -85,B 0,C 180,E1 26730.003,E2 26730.003} C_VEL
LIN {X 0,Y 54.896,Z 814.44,A -85,B 0,C 180,E1 26764.381,E2 26764.381} C_VEL
LIN {X 0,Y 72.183,Z 810.775,A -85,B 0,C 180,E1 26786.756,E2 26786.756} C_VEL
LIN {X 0,Y 73.293,Z 810.383,A -85,B 0,C 180,E1 26789.47,E2 26789.47} C_VEL
LIN {X 0,Y 72.283,Z 816.098,A -85,B 0,C 180,E1 26846.576,E2 26846.576} C_VEL
LIN {X 0,Y 58.608,Z 820.438,A -85,B 0,C 180,E1 26862.021,E2 26862.021} C_VEL
LIN {X 0,Y 47.634,Z 823.474,A -85,B 0,C 180,E1 26897.121,E2 26897.121} C_VEL
LIN {X 0,Y 45.272,Z 823.409,A -85,B 0,C 180,E1 26910.197,E2 26910.197} C_VEL
LIN {X 0,Y 42.864,Z 820.87,A -85,B 0,C 180,E1 26942.636,E2 26942.636} C_VEL
LIN {X 0,Y 57.447,Z 816.072,A -85,B 0,C 180,E1 26969.182,E2 26969.182} C_VEL
LIN {X 0,Y 59.282,Z 815.223,A -85,B 0,C 180,E1 26972.106,E2 26972.106} C_VEL
LIN {X 0,Y 71.368,Z 806.438,A -85,B 0,C 180,E1 27029.382,E2 27029.382} C_VEL
LIN {X 0,Y 70.601,Z 806.82,A -85,B 0,C 180,E1 27031.239,E2 27031.239} C_VEL
LIN {X 0,Y 50.157,Z 812.893,A -85,B 0,C 180,E1 27053.007,E2 27053.007} C_VEL
LIN {X 0,Y 41.181,Z 815.585,A -85,B 0,C 180,E1 27090.004,E2 27090.004} C_VEL
LIN {X 0,Y 48.121,Z 815.204,A -85,B 0,C 180,E1 27128.852,E2 27128.852} C_VEL
LIN {X 0,Y 62.588,Z 812.658,A -85,B 0,C 180,E1 27148.04,E2 27148.04} C_VEL
LIN {X 0,Y 64.036,Z 812.336,A -85,B 0,C 180,E1 27150.357,E2 27150.357} C_VEL
LIN {X 0,Y 62.181,Z 817.137,A -85,B 0,C 180,E1 27204.214,E2 27204.214} C_VEL
LIN {X 0,Y 60.255,Z 818,A -85,B 0,C 180,E1 27208.127,E2 27208.127} C_VEL
LIN {X 0,Y 45.846,Z 821.519,A -85,B 0,C 180,E1 27228.82,E2 27228.82} C_VEL
LIN {X 0,Y 40.151,Z 822.936,A -85,B 0,C 180,E1 27269.996,E2 27269.996} C_VEL
LIN {X 0,Y 42.864,Z 820.87,A -85,B 0,C 180,E1 27302.636,E2 27302.636} C_VEL
LIN {X 0,Y 44.383,Z 819.108,A -85,B 0,C 180,E1 27317.825,E2 27317.825} C_VEL
LIN {X 0,Y 48.402,Z 816.793,A -85,B 0,C 180,E1 27331.424,E2 27331.424} C_VEL
LIN {X 0,Y 50.501,Z 816.204,A -85,B 0,C 180,E1 27333.698,E2 27333.698} C_VEL
LIN {X 0,Y 60.515,Z 809.413,A -85,B 0,C 180,E1 27388.362,E2 27388.362} C_VEL
LIN {X 0,Y 49.128,Z 812.433,A -85,B 0,C 180,E1 27399.833,E2 27399.833} C_VEL
LIN {X 0,Y 36.579,Z 815.312,A -85,B 0,C 180,E1 27425.637,E2 27425.637} C_VEL
LIN {X 0,Y 33.296,Z 816.299,A -85,B 0,C 180,E1 27450.005,E2 27450.005} C_VEL
LIN {X 0,Y 42.213,Z 815.901,A -85,B 0,C 180,E1 27495.651,E2 27495.651} C_VEL
LIN {X 0,Y 52.598,Z 814.431,A -85,B 0,C 180,E1 27509.411,E2 27509.411} C_VEL
LIN {X 0,Y 54.167,Z 814.201,A -85,B 0,C 180,E1 27512.142,E2 27512.142} C_VEL
LIN {X 0,Y 52.852,Z 818.071,A -85,B 0,C 180,E1 27562.908,E2 27562.908} C_VEL
LIN {X 0,Y 40.087,Z 820.801,A -85,B 0,C 180,E1 27581.147,E2 27581.147} C_VEL
LIN {X 0,Y 32.204,Z 822.218,A -85,B 0,C 180,E1 27629.995,E2 27629.995} C_VEL
LIN {X 0,Y 40.136,Z 819.191,A -85,B 0,C 180,E1 27678.761,E2 27678.761} C_VEL
LIN {X 0,Y 48.402,Z 816.793,A -85,B 0,C 180,E1 27691.424,E2 27691.424} C_VEL
LIN {X 0,Y 48.695,Z 816.005,A -85,B 0,C 180,E1 27696.822,E2 27696.822} C_VEL
LIN {X 0,Y 40.696,Z 814.92,A -85,B 0,C 180,E1 27720.564,E2 27720.564} C_VEL
LIN {X 0,Y 48.952,Z 812.193,A -85,B 0,C 180,E1 27745.814,E2 27745.814} C_VEL
LIN {X 0,Y 44.503,Z 813.191,A -85,B 0,C 180,E1 27752.034,E2 27752.034} C_VEL
LIN {X 0,Y 29.578,Z 816.046,A -85,B 0,C 180,E1 27779.327,E2 27779.327} C_VEL
LIN {X 0,Y 25.388,Z 817.014,A -85,B 0,C 180,E1 27810.006,E2 27810.006} C_VEL
LIN {X 0,Y 40.728,Z 816.197,A -85,B 0,C 180,E1 27869.554,E2 27869.554} C_VEL
LIN {X 0,Y 43.871,Z 815.915,A -85,B 0,C 180,E1 27875.946,E2 27875.946} C_VEL
LIN {X 0,Y 43.31,Z 818.709,A -85,B 0,C 180,E1 27920.342,E2 27920.342} C_VEL
LIN {X 0,Y 26.356,Z 821.24,A -85,B 0,C 180,E1 27955.06,E2 27955.06} C_VEL
LIN {X 0,Y 24.256,Z 821.5,A -85,B 0,C 180,E1 27989.993,E2 27989.993} C_VEL
LIN {X 0,Y 35.298,Z 818.422,A -85,B 0,C 180,E1 28048.764,E2 28048.764} C_VEL
LIN {X 0,Y 41.267,Z 816.791,A -85,B 0,C 180,E1 28058.602,E2 28058.602} C_VEL
LIN {X 0,Y 40.696,Z 814.92,A -85,B 0,C 180,E1 28080.564,E2 28080.564} C_VEL
LIN {X 0,Y 39.563,Z 814.545,A -85,B 0,C 180,E1 28091.13,E2 28091.13} C_VEL
LIN {X 0,Y 34.027,Z 815.22,A -85,B 0,C 180,E1 28106.242,E2 28106.242} C_VEL
LIN {X 0,Y 29.618,Z 815.77,A -85,B 0,C 180,E1 28114.722,E2 28114.722} C_VEL
LIN {X 0,Y 17.499,Z 817.727,A -85,B 0,C 180,E1 28170.009,E2 28170.009} C_VEL
LIN {X 0,Y 33.093,Z 817.299,A -85,B 0,C 180,E1 28235.808,E2 28235.808} C_VEL
LIN {X 0,Y 34.358,Z 817.25,A -85,B 0,C 180,E1 28239.788,E2 28239.788} C_VEL
LIN {X 0,Y 33.454,Z 818.916,A -85,B 0,C 180,E1 28272.966,E2 28272.966} C_VEL
LIN {X 0,Y 31.806,Z 819.365,A -85,B 0,C 180,E1 28278.362,E2 28278.362} C_VEL
LIN {X 0,Y 16.291,Z 820.781,A -85,B 0,C 180,E1 28349.99,E2 28349.99} C_VEL
LIN {X 0,Y 31.738,Z 817.62,A -85,B 0,C 180,E1 28421.979,E2 28421.979} C_VEL
LIN {X 0,Y 38.257,Z 814.438,A -85,B 0,C 180,E1 28463.288,E2 28463.288} C_VEL
LIN {X 0,Y 29.618,Z 815.77,A -85,B 0,C 180,E1 28474.722,E2 28474.722} C_VEL
LIN {X 0,Y 18.83,Z 817.353,A -85,B 0,C 180,E1 28492.473,E2 28492.473} C_VEL
LIN {X 0,Y 12.943,Z 818.545,A -85,B 0,C 180,E1 28578.898,E2 28578.898} C_VEL
LIN {X 0,Y 23.318,Z 818.414,A -85,B 0,C 180,E1 28602.969,E2 28602.969} C_VEL
LIN {X 0,Y 25.023,Z 818.427,A -85,B 0,C 180,E1 28607.96,E2 28607.96} C_VEL
LIN {X 0,Y 24.661,Z 819.051,A -85,B 0,C 180,E1 28624.389,E2 28624.389} C_VEL
LIN {X 0,Y 20.294,Z 819.545,A -85,B 0,C 180,E1 28632.375,E2 28632.375} C_VEL
LIN {X 0,Y 8.299,Z 820.059,A -85,B 0,C 180,E1 28709.981,E2 28709.981} C_VEL
LIN {X 0,Y 22.59,Z 818.07,A -85,B 0,C 180,E1 28790.175,E2 28790.175} C_VEL
LIN {X 0,Y 24.649,Z 817.393,A -85,B 0,C 180,E1 28800.08,E2 28800.08} C_VEL
LIN {X 0,Y 27.112,Z 816.503,A -85,B 0,C 180,E1 28816.234,E2 28816.234} C_VEL
LIN {X 0,Y 24.407,Z 816.802,A -85,B 0,C 180,E1 28821.968,E2 28821.968} C_VEL
LIN {X 0,Y 9.59,Z 818.442,A -85,B 0,C 180,E1 28890.017,E2 28890.017} C_VEL
LIN {X 0,Y 12.943,Z 818.545,A -85,B 0,C 180,E1 28938.898,E2 28938.898} C_VEL
LIN {X 0,Y 10.844,Z 818.953,A -85,B 0,C 180,E1 28949.914,E2 28949.914} C_VEL
LIN {X 0,Y 1.118,Z 819.336,A -85,B 0,C 180,E1 28985.377,E2 28985.377} C_VEL
LIN {X 0,Y 1.884,Z 819.254,A -85,B 0,C 180,E1 29161.05,E2 29161.05} C_VEL
LIN {X 0,Y 1.696,Z 819.155,A -85,B 0,C 180,E1 29250.094,E2 29250.094} C_VEL
LIN {X 0,Y 1.118,Z 819.336,A -85,B 0,C 180,E1 29345.377,E2 29345.377} C_VEL
LIN {X 0,Y 0.974,Z 821.336,A -85,B 0,C 180,E1 29490.591,E2 29490.591} C_VEL
LIN {X 0,Y 0.974,Z 862.5,A -85,B 0,C 180,E1 29490.591,E2 29490.591} C_VEL
LIN {X 0,Y 0.974,Z 862.5,A -85,B 0,C 180,E1 29490.591,E2 29490.591}

